PROGRAM PRG_KnxLine_1
  VAR
    M1_001_401_RMA6001_MOV_ACT : FbDPT_Switch_pro;
    M1_002_401_RMA6002_MOV_ACT : FbDPT_Switch_pro;
    M1_003_406_RMA6003_MOV_ACT : FbDPT_Switch_pro;
    M1_004_407_RMA6004_MOV_ACT : FbDPT_Switch_pro;
    M1_005_408_RMA6005_MOV_ACT : FbDPT_Switch_pro;
    M1_006_409_RMA6006_MOV_ACT : FbDPT_Switch_pro;
    M1_007_409_RMA6007_MOV_ACT : FbDPT_Switch_pro;
    M1_008_409_RMA6008_MOV_ACT : FbDPT_Switch_pro;
    M1_009_464_RMA6009_MOV_ACT : FbDPT_Switch_pro;
    M1_010_464_RMA6010_MOV_ACT : FbDPT_Switch_pro;
    M1_011_415_RMA6011_MOV_ACT : FbDPT_Switch_pro;
    M1_012_422_RMA6012_MOV_ACT : FbDPT_Switch_pro;
    M1_013_422_RMA6013_MOV_ACT : FbDPT_Switch_pro;
    M1_014_426_1_RMA6014_MOV_ACT : FbDPT_Switch_pro;
    M1_015_426_2_RMA6015_MOV_ACT : FbDPT_Switch_pro;
    M1_016_426_3_RMA6016_MOV_ACT : FbDPT_Switch_pro;
    M1_017_401_RMA6001_TMP_ACT : FbDPT_Value_Temp_pro;
    M1_018_401_RMA6002_TMP_ACT : FbDPT_Value_Temp_pro;
    M1_019_406_RMA6003_TMP_ACT : FbDPT_Value_Temp_pro;
    M1_020_407_RMA6004_TMP_ACT : FbDPT_Value_Temp_pro;
    M1_021_408_RMA6005_TMP_ACT : FbDPT_Value_Temp_pro;
    M1_022_409_RMA6006_TMP_ACT : FbDPT_Value_Temp_pro;
    M1_023_409_RMA6007_TMP_ACT : FbDPT_Value_Temp_pro;
    M1_024_409_RMA6008_TMP_ACT : FbDPT_Value_Temp_pro;
    M1_025_464_RMA6009_TMP_ACT : FbDPT_Value_Temp_pro;
    M1_026_464_RMA6010_TMP_ACT : FbDPT_Value_Temp_pro;
    M1_027_415_RMA6011_TMP_ACT : FbDPT_Value_Temp_pro;
    M1_028_422_RMA6012_TMP_ACT : FbDPT_Value_Temp_pro;
    M1_029_422_RMA6013_TMP_ACT : FbDPT_Value_Temp_pro;
    M1_030_426_1_RMA6014_TMP_ACT : FbDPT_Value_Temp_pro;
    M1_031_426_2_RMA6015_TMP_ACT : FbDPT_Value_Temp_pro;
    M1_032_426_3_RMA6016_TMP_ACT : FbDPT_Value_Temp_pro;
    M1_033_401_RMA6001_CO2_ACT : FbDPT_Value_AirQuality_pro;
    M1_034_401_RMA6002_CO2_ACT : FbDPT_Value_AirQuality_pro;
    M1_035_406_RMA6003_CO2_ACT : FbDPT_Value_AirQuality_pro;
    M1_036_407_RMA6004_CO2_ACT : FbDPT_Value_AirQuality_pro;
    M1_037_408_RMA6005_CO2_ACT : FbDPT_Value_AirQuality_pro;
    M1_038_409_RMA6006_CO2_ACT : FbDPT_Value_AirQuality_pro;
    M1_039_409_RMA6007_CO2_ACT : FbDPT_Value_AirQuality_pro;
    M1_040_409_RMA6008_CO2_ACT : FbDPT_Value_AirQuality_pro;
    M1_041_464_RMA6009_CO2_ACT : FbDPT_Value_AirQuality_pro;
    M1_042_464_RMA6010_CO2_ACT : FbDPT_Value_AirQuality_pro;
    M1_043_415_RMA6011_CO2_ACT : FbDPT_Value_AirQuality_pro;
    M1_044_422_RMA6012_CO2_ACT : FbDPT_Value_AirQuality_pro;
    M1_045_422_RMA6013_CO2_ACT : FbDPT_Value_AirQuality_pro;
    M1_046_426_1_RMA6014_CO2_ACT : FbDPT_Value_AirQuality_pro;
    M1_047_426_2_RMA6015_CO2_ACT : FbDPT_Value_AirQuality_pro;
    M1_048_426_3_RMA6016_CO2_ACT : FbDPT_Value_AirQuality_pro;
    M1_049_401_KAB6001_CV : FbDPT_Scaling_pro;
    M1_050_401_KAB6001_POS_ACT : FbDPT_Scaling_pro;
    M1_051_401_KAB6002_CV : FbDPT_Scaling_pro;
    M1_052_401_KAB6002_POS_ACT : FbDPT_Scaling_pro;
    M1_053_401_KAB6003_CV : FbDPT_Scaling_pro;
    M1_054_401_KAB6003_POS_ACT : FbDPT_Scaling_pro;
    M1_055_401_KAB6004_CV : FbDPT_Scaling_pro;
    M1_056_401_KAB6004_POS_ACT : FbDPT_Scaling_pro;
    M1_057_401_KAB6005_CV : FbDPT_Scaling_pro;
    M1_058_401_KAB6005_POS_ACT : FbDPT_Scaling_pro;
    M1_059_406_KAB6006_CV : FbDPT_Scaling_pro;
    M1_060_406_KAB6006_POS_ACT : FbDPT_Scaling_pro;
    M1_061_406_KAB6007_CV : FbDPT_Scaling_pro;
    M1_062_406_KAB6007_POS_ACT : FbDPT_Scaling_pro;
    M1_063_407_KAB6008_CV : FbDPT_Scaling_pro;
    M1_064_407_KAB6008_POS_ACT : FbDPT_Scaling_pro;
    M1_065_407_KAB6009_CV : FbDPT_Scaling_pro;
    M1_066_407_KAB6009_POS_ACT : FbDPT_Scaling_pro;
    M1_067_408_KAB6010_CV : FbDPT_Scaling_pro;
    M1_068_408_KAB6010_POS_ACT : FbDPT_Scaling_pro;
    M1_069_409_KAB6011_CV : FbDPT_Scaling_pro;
    M1_070_409_KAB6011_POS_ACT : FbDPT_Scaling_pro;
    M1_071_409_KAB6012_CV : FbDPT_Scaling_pro;
    M1_072_409_KAB6012_POS_ACT : FbDPT_Scaling_pro;
    M1_073_409_KAB6013_CV : FbDPT_Scaling_pro;
    M1_074_409_KAB6013_POS_ACT : FbDPT_Scaling_pro;
    M1_075_409_KAB6014_CV : FbDPT_Scaling_pro;
    M1_076_409_KAB6014_POS_ACT : FbDPT_Scaling_pro;
    M1_077_409_KAB6015_CV : FbDPT_Scaling_pro;
    M1_078_409_KAB6015_POS_ACT : FbDPT_Scaling_pro;
    M1_079_409_KAB6016_CV : FbDPT_Scaling_pro;
    M1_080_409_KAB6016_POS_ACT : FbDPT_Scaling_pro;
    M1_081_409_KAB6017_CV : FbDPT_Scaling_pro;
    M1_082_409_KAB6017_POS_ACT : FbDPT_Scaling_pro;
    M1_083_464_KAB6018_CV : FbDPT_Scaling_pro;
    M1_084_464_KAB6018_POS_ACT : FbDPT_Scaling_pro;
    M1_085_464_KAB6019_CV : FbDPT_Scaling_pro;
    M1_086_464_KAB6019_POS_ACT : FbDPT_Scaling_pro;
    M1_087_464_KAB6020_CV : FbDPT_Scaling_pro;
    M1_088_464_KAB6020_POS_ACT : FbDPT_Scaling_pro;
    M1_089_464_KAB6021_CV : FbDPT_Scaling_pro;
    M1_090_464_KAB6021_POS_ACT : FbDPT_Scaling_pro;
    M1_091_415_KAB6022_CV : FbDPT_Scaling_pro;
    M1_092_415_KAB6022_POS_ACT : FbDPT_Scaling_pro;
    M1_093_415_KAB6023_CV : FbDPT_Scaling_pro;
    M1_094_415_KAB6023_POS_ACT : FbDPT_Scaling_pro;
    M1_095_422_KAB6024_CV : FbDPT_Scaling_pro;
    M1_096_422_KAB6024_POS_ACT : FbDPT_Scaling_pro;
    M1_097_422_KAB6025_CV : FbDPT_Scaling_pro;
    M1_098_422_KAB6025_POS_ACT : FbDPT_Scaling_pro;
    M1_099_422_KAB6026_CV : FbDPT_Scaling_pro;
    M1_100_422_KAB6026_POS_ACT : FbDPT_Scaling_pro;
    M1_101_422_KAB6027_CV : FbDPT_Scaling_pro;
    M1_102_422_KAB6027_POS_ACT : FbDPT_Scaling_pro;
    M1_103_422_KAB6028_CV : FbDPT_Scaling_pro;
    M1_104_422_KAB6028_POS_ACT : FbDPT_Scaling_pro;
    M1_105_426_1_KAB6029_CV : FbDPT_Scaling_pro;
    M1_106_426_1_KAB6029_POS_ACT : FbDPT_Scaling_pro;
    M1_107_426_2_KAB6030_CV : FbDPT_Scaling_pro;
    M1_108_426_2_KAB6030_POS_ACT : FbDPT_Scaling_pro;
    M1_109_426_3_KAB6031_CV : FbDPT_Scaling_pro;
    M1_110_426_3_KAB6031_POS_ACT : FbDPT_Scaling_pro;
  END_VAR

                
    
        M1_001_401_RMA6001_MOV_ACT(
            bPortKNX      := 1, 
            dwIndex_DPT   := 1, 
            typDPT        := PersistentVars.typDPT[1][1]
        );

        
        M1_002_401_RMA6002_MOV_ACT(
            bPortKNX      := 1, 
            dwIndex_DPT   := 2, 
            typDPT        := PersistentVars.typDPT[1][2]
        );

        
        M1_003_406_RMA6003_MOV_ACT(
            bPortKNX      := 1, 
            dwIndex_DPT   := 3, 
            typDPT        := PersistentVars.typDPT[1][3]
        );

        
        M1_004_407_RMA6004_MOV_ACT(
            bPortKNX      := 1, 
            dwIndex_DPT   := 4, 
            typDPT        := PersistentVars.typDPT[1][4]
        );

        
        M1_005_408_RMA6005_MOV_ACT(
            bPortKNX      := 1, 
            dwIndex_DPT   := 5, 
            typDPT        := PersistentVars.typDPT[1][5]
        );

        
        M1_006_409_RMA6006_MOV_ACT(
            bPortKNX      := 1, 
            dwIndex_DPT   := 6, 
            typDPT        := PersistentVars.typDPT[1][6]
        );

        
        M1_007_409_RMA6007_MOV_ACT(
            bPortKNX      := 1, 
            dwIndex_DPT   := 7, 
            typDPT        := PersistentVars.typDPT[1][7]
        );

        
        M1_008_409_RMA6008_MOV_ACT(
            bPortKNX      := 1, 
            dwIndex_DPT   := 8, 
            typDPT        := PersistentVars.typDPT[1][8]
        );

        
        M1_009_464_RMA6009_MOV_ACT(
            bPortKNX      := 1, 
            dwIndex_DPT   := 9, 
            typDPT        := PersistentVars.typDPT[1][9]
        );

        
        M1_010_464_RMA6010_MOV_ACT(
            bPortKNX      := 1, 
            dwIndex_DPT   := 10, 
            typDPT        := PersistentVars.typDPT[1][10]
        );

        
        M1_011_415_RMA6011_MOV_ACT(
            bPortKNX      := 1, 
            dwIndex_DPT   := 11, 
            typDPT        := PersistentVars.typDPT[1][11]
        );

        
        M1_012_422_RMA6012_MOV_ACT(
            bPortKNX      := 1, 
            dwIndex_DPT   := 12, 
            typDPT        := PersistentVars.typDPT[1][12]
        );

        
        M1_013_422_RMA6013_MOV_ACT(
            bPortKNX      := 1, 
            dwIndex_DPT   := 13, 
            typDPT        := PersistentVars.typDPT[1][13]
        );

        
        M1_014_426_1_RMA6014_MOV_ACT(
            bPortKNX      := 1, 
            dwIndex_DPT   := 14, 
            typDPT        := PersistentVars.typDPT[1][14]
        );

        
        M1_015_426_2_RMA6015_MOV_ACT(
            bPortKNX      := 1, 
            dwIndex_DPT   := 15, 
            typDPT        := PersistentVars.typDPT[1][15]
        );

        
        M1_016_426_3_RMA6016_MOV_ACT(
            bPortKNX      := 1, 
            dwIndex_DPT   := 16, 
            typDPT        := PersistentVars.typDPT[1][16]
        );

        
        M1_017_401_RMA6001_TMP_ACT(
            bPortKNX      := 1,
            dwIndex_DPT   := 17,
            typDPT        := PersistentVars.typDPT[1][17],
            xUpdate_PLC   => ,
            xTimeOut      => 
        );

        
                                    
        C_5640_501_06_RMA6001_A1_R0401.xIn := M1_017_401_RMA6001_TMP_ACT.xTimeOut;
                                    
        M1_018_401_RMA6002_TMP_ACT(
            bPortKNX      := 1,
            dwIndex_DPT   := 18,
            typDPT        := PersistentVars.typDPT[1][18],
            xUpdate_PLC   => ,
            xTimeOut      => 
        );

        
                                    
        C_5640_501_06_RMA6002_A1_R0401.xIn := M1_018_401_RMA6002_TMP_ACT.xTimeOut;
                                    
        M1_019_406_RMA6003_TMP_ACT(
            bPortKNX      := 1,
            dwIndex_DPT   := 19,
            typDPT        := PersistentVars.typDPT[1][19],
            xUpdate_PLC   => ,
            xTimeOut      => 
        );

        
                                    
        C_5640_501_06_RMA6003_A1_R0406.xIn := M1_019_406_RMA6003_TMP_ACT.xTimeOut;
                                    
        M1_020_407_RMA6004_TMP_ACT(
            bPortKNX      := 1,
            dwIndex_DPT   := 20,
            typDPT        := PersistentVars.typDPT[1][20],
            xUpdate_PLC   => ,
            xTimeOut      => 
        );

        
                                    
        C_5640_501_06_RMA6004_A1_R0407.xIn := M1_020_407_RMA6004_TMP_ACT.xTimeOut;
                                    
        M1_021_408_RMA6005_TMP_ACT(
            bPortKNX      := 1,
            dwIndex_DPT   := 21,
            typDPT        := PersistentVars.typDPT[1][21],
            xUpdate_PLC   => ,
            xTimeOut      => 
        );

        
                                    
        C_5640_501_06_RMA6005_A1_R0408.xIn := M1_021_408_RMA6005_TMP_ACT.xTimeOut;
                                    
        M1_022_409_RMA6006_TMP_ACT(
            bPortKNX      := 1,
            dwIndex_DPT   := 22,
            typDPT        := PersistentVars.typDPT[1][22],
            xUpdate_PLC   => ,
            xTimeOut      => 
        );

        
                                    
        C_5640_501_06_RMA6006_A1_R0409.xIn := M1_022_409_RMA6006_TMP_ACT.xTimeOut;
                                    
        M1_023_409_RMA6007_TMP_ACT(
            bPortKNX      := 1,
            dwIndex_DPT   := 23,
            typDPT        := PersistentVars.typDPT[1][23],
            xUpdate_PLC   => ,
            xTimeOut      => 
        );

        
                                    
        C_5640_501_06_RMA6007_A1_R0409.xIn := M1_023_409_RMA6007_TMP_ACT.xTimeOut;
                                    
        M1_024_409_RMA6008_TMP_ACT(
            bPortKNX      := 1,
            dwIndex_DPT   := 24,
            typDPT        := PersistentVars.typDPT[1][24],
            xUpdate_PLC   => ,
            xTimeOut      => 
        );

        
                                    
        C_5640_501_06_RMA6008_A1_R0409.xIn := M1_024_409_RMA6008_TMP_ACT.xTimeOut;
                                    
        M1_025_464_RMA6009_TMP_ACT(
            bPortKNX      := 1,
            dwIndex_DPT   := 25,
            typDPT        := PersistentVars.typDPT[1][25],
            xUpdate_PLC   => ,
            xTimeOut      => 
        );

        
                                    
        C_5640_501_06_RMA6009_A1_R0464.xIn := M1_025_464_RMA6009_TMP_ACT.xTimeOut;
                                    
        M1_026_464_RMA6010_TMP_ACT(
            bPortKNX      := 1,
            dwIndex_DPT   := 26,
            typDPT        := PersistentVars.typDPT[1][26],
            xUpdate_PLC   => ,
            xTimeOut      => 
        );

        
                                    
        C_5640_501_06_RMA6010_A1_R0464.xIn := M1_026_464_RMA6010_TMP_ACT.xTimeOut;
                                    
        M1_027_415_RMA6011_TMP_ACT(
            bPortKNX      := 1,
            dwIndex_DPT   := 27,
            typDPT        := PersistentVars.typDPT[1][27],
            xUpdate_PLC   => ,
            xTimeOut      => 
        );

        
                                    
        C_5640_501_06_RMA6011_A1_R0415.xIn := M1_027_415_RMA6011_TMP_ACT.xTimeOut;
                                    
        M1_028_422_RMA6012_TMP_ACT(
            bPortKNX      := 1,
            dwIndex_DPT   := 28,
            typDPT        := PersistentVars.typDPT[1][28],
            xUpdate_PLC   => ,
            xTimeOut      => 
        );

        
                                    
        C_5640_501_06_RMA6012_A1_R0422.xIn := M1_028_422_RMA6012_TMP_ACT.xTimeOut;
                                    
        M1_029_422_RMA6013_TMP_ACT(
            bPortKNX      := 1,
            dwIndex_DPT   := 29,
            typDPT        := PersistentVars.typDPT[1][29],
            xUpdate_PLC   => ,
            xTimeOut      => 
        );

        
                                    
        C_5640_501_06_RMA6013_A1_R0422.xIn := M1_029_422_RMA6013_TMP_ACT.xTimeOut;
                                    
        M1_030_426_1_RMA6014_TMP_ACT(
            bPortKNX      := 1,
            dwIndex_DPT   := 30,
            typDPT        := PersistentVars.typDPT[1][30],
            xUpdate_PLC   => ,
            xTimeOut      => 
        );

        
                                    
        C_5640_501_06_RMA6014_A1_R0426_1.xIn := M1_030_426_1_RMA6014_TMP_ACT.xTimeOut;
                                    
        M1_031_426_2_RMA6015_TMP_ACT(
            bPortKNX      := 1,
            dwIndex_DPT   := 31,
            typDPT        := PersistentVars.typDPT[1][31],
            xUpdate_PLC   => ,
            xTimeOut      => 
        );

        
                                    
        C_5640_501_06_RMA6015_A1_R0426_2.xIn := M1_031_426_2_RMA6015_TMP_ACT.xTimeOut;
                                    
        M1_032_426_3_RMA6016_TMP_ACT(
            bPortKNX      := 1,
            dwIndex_DPT   := 32,
            typDPT        := PersistentVars.typDPT[1][32],
            xUpdate_PLC   => ,
            xTimeOut      => 
        );

        
                                    
        C_5640_501_06_RMA6016_A1_R0426_3.xIn := M1_032_426_3_RMA6016_TMP_ACT.xTimeOut;
                                    
        M1_033_401_RMA6001_CO2_ACT(
            bPortKNX      := 1,
            dwIndex_DPT   := 33,
            typDPT        := PersistentVars.typDPT[1][33],
            xUpdate_PLC   => ,
            xTimeOut      => 
        );

        
        M1_034_401_RMA6002_CO2_ACT(
            bPortKNX      := 1,
            dwIndex_DPT   := 34,
            typDPT        := PersistentVars.typDPT[1][34],
            xUpdate_PLC   => ,
            xTimeOut      => 
        );

        
        M1_035_406_RMA6003_CO2_ACT(
            bPortKNX      := 1,
            dwIndex_DPT   := 35,
            typDPT        := PersistentVars.typDPT[1][35],
            xUpdate_PLC   => ,
            xTimeOut      => 
        );

        
        M1_036_407_RMA6004_CO2_ACT(
            bPortKNX      := 1,
            dwIndex_DPT   := 36,
            typDPT        := PersistentVars.typDPT[1][36],
            xUpdate_PLC   => ,
            xTimeOut      => 
        );

        
        M1_037_408_RMA6005_CO2_ACT(
            bPortKNX      := 1,
            dwIndex_DPT   := 37,
            typDPT        := PersistentVars.typDPT[1][37],
            xUpdate_PLC   => ,
            xTimeOut      => 
        );

        
        M1_038_409_RMA6006_CO2_ACT(
            bPortKNX      := 1,
            dwIndex_DPT   := 38,
            typDPT        := PersistentVars.typDPT[1][38],
            xUpdate_PLC   => ,
            xTimeOut      => 
        );

        
        M1_039_409_RMA6007_CO2_ACT(
            bPortKNX      := 1,
            dwIndex_DPT   := 39,
            typDPT        := PersistentVars.typDPT[1][39],
            xUpdate_PLC   => ,
            xTimeOut      => 
        );

        
        M1_040_409_RMA6008_CO2_ACT(
            bPortKNX      := 1,
            dwIndex_DPT   := 40,
            typDPT        := PersistentVars.typDPT[1][40],
            xUpdate_PLC   => ,
            xTimeOut      => 
        );

        
        M1_041_464_RMA6009_CO2_ACT(
            bPortKNX      := 1,
            dwIndex_DPT   := 41,
            typDPT        := PersistentVars.typDPT[1][41],
            xUpdate_PLC   => ,
            xTimeOut      => 
        );

        
        M1_042_464_RMA6010_CO2_ACT(
            bPortKNX      := 1,
            dwIndex_DPT   := 42,
            typDPT        := PersistentVars.typDPT[1][42],
            xUpdate_PLC   => ,
            xTimeOut      => 
        );

        
        M1_043_415_RMA6011_CO2_ACT(
            bPortKNX      := 1,
            dwIndex_DPT   := 43,
            typDPT        := PersistentVars.typDPT[1][43],
            xUpdate_PLC   => ,
            xTimeOut      => 
        );

        
        M1_044_422_RMA6012_CO2_ACT(
            bPortKNX      := 1,
            dwIndex_DPT   := 44,
            typDPT        := PersistentVars.typDPT[1][44],
            xUpdate_PLC   => ,
            xTimeOut      => 
        );

        
        M1_045_422_RMA6013_CO2_ACT(
            bPortKNX      := 1,
            dwIndex_DPT   := 45,
            typDPT        := PersistentVars.typDPT[1][45],
            xUpdate_PLC   => ,
            xTimeOut      => 
        );

        
        M1_046_426_1_RMA6014_CO2_ACT(
            bPortKNX      := 1,
            dwIndex_DPT   := 46,
            typDPT        := PersistentVars.typDPT[1][46],
            xUpdate_PLC   => ,
            xTimeOut      => 
        );

        
        M1_047_426_2_RMA6015_CO2_ACT(
            bPortKNX      := 1,
            dwIndex_DPT   := 47,
            typDPT        := PersistentVars.typDPT[1][47],
            xUpdate_PLC   => ,
            xTimeOut      => 
        );

        
        M1_048_426_3_RMA6016_CO2_ACT(
            bPortKNX      := 1,
            dwIndex_DPT   := 48,
            typDPT        := PersistentVars.typDPT[1][48],
            xUpdate_PLC   => ,
            xTimeOut      => 
        );

        
        M1_049_401_KAB6001_CV(
            bPortKNX		  := 1, 
            dwIndex_DPT		:= 49, 
            typDPT			  := PersistentVars.typDPT[1][49],
            xUpdate_KNX		:= PRG_KnxMaster.updateHeat, 
        );

        M1_049_401_KAB6001_CV.rValue_IN := GVL_ClimateControl.typClimateControllerInterfaceRoom401.actuators.heating.controlledVariable;        
         
        M1_050_401_KAB6001_POS_ACT(
            bPortKNX		   := 1, 
            dwIndex_DPT		:= 50, 
            typDPT			  := PersistentVars.typDPT[1][50], 
        );

        
                                    
        C_5640_501_06_KAB6001_A1_R0401.xIn := M1_050_401_KAB6001_POS_ACT.xTimeOut;
                                    
        M1_051_401_KAB6002_CV(
            bPortKNX		  := 1, 
            dwIndex_DPT		:= 51, 
            typDPT			  := PersistentVars.typDPT[1][51],
            xUpdate_KNX		:= PRG_KnxMaster.updateHeat, 
        );

        M1_051_401_KAB6002_CV.rValue_IN := GVL_ClimateControl.typClimateControllerInterfaceRoom401.actuators.heating.controlledVariable;        
         
        M1_052_401_KAB6002_POS_ACT(
            bPortKNX		   := 1, 
            dwIndex_DPT		:= 52, 
            typDPT			  := PersistentVars.typDPT[1][52], 
        );

        
                                    
        C_5640_501_06_KAB6002_A1_R0401.xIn := M1_052_401_KAB6002_POS_ACT.xTimeOut;
                                    
        M1_053_401_KAB6003_CV(
            bPortKNX		  := 1, 
            dwIndex_DPT		:= 53, 
            typDPT			  := PersistentVars.typDPT[1][53],
            xUpdate_KNX		:= PRG_KnxMaster.updateHeat, 
        );

        M1_053_401_KAB6003_CV.rValue_IN := GVL_ClimateControl.typClimateControllerInterfaceRoom401.actuators.heating.controlledVariable;        
         
        M1_054_401_KAB6003_POS_ACT(
            bPortKNX		   := 1, 
            dwIndex_DPT		:= 54, 
            typDPT			  := PersistentVars.typDPT[1][54], 
        );

        
                                    
        C_5640_501_06_KAB6003_A1_R0401.xIn := M1_054_401_KAB6003_POS_ACT.xTimeOut;
                                    
        M1_055_401_KAB6004_CV(
            bPortKNX		  := 1, 
            dwIndex_DPT		:= 55, 
            typDPT			  := PersistentVars.typDPT[1][55],
            xUpdate_KNX		:= PRG_KnxMaster.updateHeat, 
        );

        M1_055_401_KAB6004_CV.rValue_IN := GVL_ClimateControl.typClimateControllerInterfaceRoom401.actuators.heating.controlledVariable;        
         
        M1_056_401_KAB6004_POS_ACT(
            bPortKNX		   := 1, 
            dwIndex_DPT		:= 56, 
            typDPT			  := PersistentVars.typDPT[1][56], 
        );

        
                                    
        C_5640_501_06_KAB6004_A1_R0401.xIn := M1_056_401_KAB6004_POS_ACT.xTimeOut;
                                    
        M1_057_401_KAB6005_CV(
            bPortKNX		  := 1, 
            dwIndex_DPT		:= 57, 
            typDPT			  := PersistentVars.typDPT[1][57],
            xUpdate_KNX		:= PRG_KnxMaster.updateHeat, 
        );

        M1_057_401_KAB6005_CV.rValue_IN := GVL_ClimateControl.typClimateControllerInterfaceRoom401.actuators.heating.controlledVariable;        
         
        M1_058_401_KAB6005_POS_ACT(
            bPortKNX		   := 1, 
            dwIndex_DPT		:= 58, 
            typDPT			  := PersistentVars.typDPT[1][58], 
        );

        
                                    
        C_5640_501_06_KAB6005_A1_R0401.xIn := M1_058_401_KAB6005_POS_ACT.xTimeOut;
                                    
        M1_059_406_KAB6006_CV(
            bPortKNX		  := 1, 
            dwIndex_DPT		:= 59, 
            typDPT			  := PersistentVars.typDPT[1][59],
            xUpdate_KNX		:= PRG_KnxMaster.updateHeat, 
        );

        M1_059_406_KAB6006_CV.rValue_IN := GVL_ClimateControl.typClimateControllerInterfaceRoom406.actuators.heating.controlledVariable;        
         
        M1_060_406_KAB6006_POS_ACT(
            bPortKNX		   := 1, 
            dwIndex_DPT		:= 60, 
            typDPT			  := PersistentVars.typDPT[1][60], 
        );

        
                                    
        C_5640_501_06_KAB6006_A1_R0406.xIn := M1_060_406_KAB6006_POS_ACT.xTimeOut;
                                    
        M1_061_406_KAB6007_CV(
            bPortKNX		  := 1, 
            dwIndex_DPT		:= 61, 
            typDPT			  := PersistentVars.typDPT[1][61],
            xUpdate_KNX		:= PRG_KnxMaster.updateHeat, 
        );

        M1_061_406_KAB6007_CV.rValue_IN := GVL_ClimateControl.typClimateControllerInterfaceRoom406.actuators.heating.controlledVariable;        
         
        M1_062_406_KAB6007_POS_ACT(
            bPortKNX		   := 1, 
            dwIndex_DPT		:= 62, 
            typDPT			  := PersistentVars.typDPT[1][62], 
        );

        
                                    
        C_5640_501_06_KAB6007_A1_R0406.xIn := M1_062_406_KAB6007_POS_ACT.xTimeOut;
                                    
        M1_063_407_KAB6008_CV(
            bPortKNX		  := 1, 
            dwIndex_DPT		:= 63, 
            typDPT			  := PersistentVars.typDPT[1][63],
            xUpdate_KNX		:= PRG_KnxMaster.updateHeat, 
        );

        M1_063_407_KAB6008_CV.rValue_IN := GVL_ClimateControl.typClimateControllerInterfaceRoom407.actuators.heating.controlledVariable;        
         
        M1_064_407_KAB6008_POS_ACT(
            bPortKNX		   := 1, 
            dwIndex_DPT		:= 64, 
            typDPT			  := PersistentVars.typDPT[1][64], 
        );

        
                                    
        C_5640_501_06_KAB6008_A1_R0407.xIn := M1_064_407_KAB6008_POS_ACT.xTimeOut;
                                    
        M1_065_407_KAB6009_CV(
            bPortKNX		  := 1, 
            dwIndex_DPT		:= 65, 
            typDPT			  := PersistentVars.typDPT[1][65],
            xUpdate_KNX		:= PRG_KnxMaster.updateHeat, 
        );

        M1_065_407_KAB6009_CV.rValue_IN := GVL_ClimateControl.typClimateControllerInterfaceRoom407.actuators.heating.controlledVariable;        
         
        M1_066_407_KAB6009_POS_ACT(
            bPortKNX		   := 1, 
            dwIndex_DPT		:= 66, 
            typDPT			  := PersistentVars.typDPT[1][66], 
        );

        
                                    
        C_5640_501_06_KAB6009_A1_R0407.xIn := M1_066_407_KAB6009_POS_ACT.xTimeOut;
                                    
        M1_067_408_KAB6010_CV(
            bPortKNX		  := 1, 
            dwIndex_DPT		:= 67, 
            typDPT			  := PersistentVars.typDPT[1][67],
            xUpdate_KNX		:= PRG_KnxMaster.updateHeat, 
        );

        M1_067_408_KAB6010_CV.rValue_IN := GVL_ClimateControl.typClimateControllerInterfaceRoom408.actuators.heating.controlledVariable;        
         
        M1_068_408_KAB6010_POS_ACT(
            bPortKNX		   := 1, 
            dwIndex_DPT		:= 68, 
            typDPT			  := PersistentVars.typDPT[1][68], 
        );

        
                                    
        C_5640_501_06_KAB6010_A1_R0408.xIn := M1_068_408_KAB6010_POS_ACT.xTimeOut;
                                    
        M1_069_409_KAB6011_CV(
            bPortKNX		  := 1, 
            dwIndex_DPT		:= 69, 
            typDPT			  := PersistentVars.typDPT[1][69],
            xUpdate_KNX		:= PRG_KnxMaster.updateHeat, 
        );

        M1_069_409_KAB6011_CV.rValue_IN := GVL_ClimateControl.typClimateControllerInterfaceRoom409.actuators.heating.controlledVariable;        
         
        M1_070_409_KAB6011_POS_ACT(
            bPortKNX		   := 1, 
            dwIndex_DPT		:= 70, 
            typDPT			  := PersistentVars.typDPT[1][70], 
        );

        
                                    
        C_5640_501_06_KAB6011_A1_R0409.xIn := M1_070_409_KAB6011_POS_ACT.xTimeOut;
                                    
        M1_071_409_KAB6012_CV(
            bPortKNX		  := 1, 
            dwIndex_DPT		:= 71, 
            typDPT			  := PersistentVars.typDPT[1][71],
            xUpdate_KNX		:= PRG_KnxMaster.updateHeat, 
        );

        M1_071_409_KAB6012_CV.rValue_IN := GVL_ClimateControl.typClimateControllerInterfaceRoom409.actuators.heating.controlledVariable;        
         
        M1_072_409_KAB6012_POS_ACT(
            bPortKNX		   := 1, 
            dwIndex_DPT		:= 72, 
            typDPT			  := PersistentVars.typDPT[1][72], 
        );

        
                                    
        C_5640_501_06_KAB6012_A1_R0409.xIn := M1_072_409_KAB6012_POS_ACT.xTimeOut;
                                    
        M1_073_409_KAB6013_CV(
            bPortKNX		  := 1, 
            dwIndex_DPT		:= 73, 
            typDPT			  := PersistentVars.typDPT[1][73],
            xUpdate_KNX		:= PRG_KnxMaster.updateHeat, 
        );

        M1_073_409_KAB6013_CV.rValue_IN := GVL_ClimateControl.typClimateControllerInterfaceRoom409.actuators.heating.controlledVariable;        
         
        M1_074_409_KAB6013_POS_ACT(
            bPortKNX		   := 1, 
            dwIndex_DPT		:= 74, 
            typDPT			  := PersistentVars.typDPT[1][74], 
        );

        
                                    
        C_5640_501_06_KAB6013_A1_R0409.xIn := M1_074_409_KAB6013_POS_ACT.xTimeOut;
                                    
        M1_075_409_KAB6014_CV(
            bPortKNX		  := 1, 
            dwIndex_DPT		:= 75, 
            typDPT			  := PersistentVars.typDPT[1][75],
            xUpdate_KNX		:= PRG_KnxMaster.updateHeat, 
        );

        M1_075_409_KAB6014_CV.rValue_IN := GVL_ClimateControl.typClimateControllerInterfaceRoom409.actuators.heating.controlledVariable;        
         
        M1_076_409_KAB6014_POS_ACT(
            bPortKNX		   := 1, 
            dwIndex_DPT		:= 76, 
            typDPT			  := PersistentVars.typDPT[1][76], 
        );

        
                                    
        C_5640_501_06_KAB6014_A1_R0409.xIn := M1_076_409_KAB6014_POS_ACT.xTimeOut;
                                    
        M1_077_409_KAB6015_CV(
            bPortKNX		  := 1, 
            dwIndex_DPT		:= 77, 
            typDPT			  := PersistentVars.typDPT[1][77],
            xUpdate_KNX		:= PRG_KnxMaster.updateHeat, 
        );

        M1_077_409_KAB6015_CV.rValue_IN := GVL_ClimateControl.typClimateControllerInterfaceRoom409.actuators.heating.controlledVariable;        
         
        M1_078_409_KAB6015_POS_ACT(
            bPortKNX		   := 1, 
            dwIndex_DPT		:= 78, 
            typDPT			  := PersistentVars.typDPT[1][78], 
        );

        
                                    
        C_5640_501_06_KAB6015_A1_R0409.xIn := M1_078_409_KAB6015_POS_ACT.xTimeOut;
                                    
        M1_079_409_KAB6016_CV(
            bPortKNX		  := 1, 
            dwIndex_DPT		:= 79, 
            typDPT			  := PersistentVars.typDPT[1][79],
            xUpdate_KNX		:= PRG_KnxMaster.updateHeat, 
        );

        M1_079_409_KAB6016_CV.rValue_IN := GVL_ClimateControl.typClimateControllerInterfaceRoom409.actuators.heating.controlledVariable;        
         
        M1_080_409_KAB6016_POS_ACT(
            bPortKNX		   := 1, 
            dwIndex_DPT		:= 80, 
            typDPT			  := PersistentVars.typDPT[1][80], 
        );

        
                                    
        C_5640_501_06_KAB6016_A1_R0409.xIn := M1_080_409_KAB6016_POS_ACT.xTimeOut;
                                    
        M1_081_409_KAB6017_CV(
            bPortKNX		  := 1, 
            dwIndex_DPT		:= 81, 
            typDPT			  := PersistentVars.typDPT[1][81],
            xUpdate_KNX		:= PRG_KnxMaster.updateHeat, 
        );

        M1_081_409_KAB6017_CV.rValue_IN := GVL_ClimateControl.typClimateControllerInterfaceRoom409.actuators.heating.controlledVariable;        
         
        M1_082_409_KAB6017_POS_ACT(
            bPortKNX		   := 1, 
            dwIndex_DPT		:= 82, 
            typDPT			  := PersistentVars.typDPT[1][82], 
        );

        
                                    
        C_5640_501_06_KAB6017_A1_R0409.xIn := M1_082_409_KAB6017_POS_ACT.xTimeOut;
                                    
        M1_083_464_KAB6018_CV(
            bPortKNX		  := 1, 
            dwIndex_DPT		:= 83, 
            typDPT			  := PersistentVars.typDPT[1][83],
            xUpdate_KNX		:= PRG_KnxMaster.updateHeat, 
        );

        M1_083_464_KAB6018_CV.rValue_IN := GVL_ClimateControl.typClimateControllerInterfaceRoom464.actuators.heating.controlledVariable;        
         
        M1_084_464_KAB6018_POS_ACT(
            bPortKNX		   := 1, 
            dwIndex_DPT		:= 84, 
            typDPT			  := PersistentVars.typDPT[1][84], 
        );

        
                                    
        C_5640_501_06_KAB6018_A1_R0464.xIn := M1_084_464_KAB6018_POS_ACT.xTimeOut;
                                    
        M1_085_464_KAB6019_CV(
            bPortKNX		  := 1, 
            dwIndex_DPT		:= 85, 
            typDPT			  := PersistentVars.typDPT[1][85],
            xUpdate_KNX		:= PRG_KnxMaster.updateHeat, 
        );

        M1_085_464_KAB6019_CV.rValue_IN := GVL_ClimateControl.typClimateControllerInterfaceRoom464.actuators.heating.controlledVariable;        
         
        M1_086_464_KAB6019_POS_ACT(
            bPortKNX		   := 1, 
            dwIndex_DPT		:= 86, 
            typDPT			  := PersistentVars.typDPT[1][86], 
        );

        
                                    
        C_5640_501_06_KAB6019_A1_R0464.xIn := M1_086_464_KAB6019_POS_ACT.xTimeOut;
                                    
        M1_087_464_KAB6020_CV(
            bPortKNX		  := 1, 
            dwIndex_DPT		:= 87, 
            typDPT			  := PersistentVars.typDPT[1][87],
            xUpdate_KNX		:= PRG_KnxMaster.updateHeat, 
        );

        M1_087_464_KAB6020_CV.rValue_IN := GVL_ClimateControl.typClimateControllerInterfaceRoom464.actuators.heating.controlledVariable;        
         
        M1_088_464_KAB6020_POS_ACT(
            bPortKNX		   := 1, 
            dwIndex_DPT		:= 88, 
            typDPT			  := PersistentVars.typDPT[1][88], 
        );

        
                                    
        C_5640_501_06_KAB6020_A1_R0464.xIn := M1_088_464_KAB6020_POS_ACT.xTimeOut;
                                    
        M1_089_464_KAB6021_CV(
            bPortKNX		  := 1, 
            dwIndex_DPT		:= 89, 
            typDPT			  := PersistentVars.typDPT[1][89],
            xUpdate_KNX		:= PRG_KnxMaster.updateHeat, 
        );

        M1_089_464_KAB6021_CV.rValue_IN := GVL_ClimateControl.typClimateControllerInterfaceRoom464.actuators.heating.controlledVariable;        
         
        M1_090_464_KAB6021_POS_ACT(
            bPortKNX		   := 1, 
            dwIndex_DPT		:= 90, 
            typDPT			  := PersistentVars.typDPT[1][90], 
        );

        
                                    
        C_5640_501_06_KAB6021_A1_R0464.xIn := M1_090_464_KAB6021_POS_ACT.xTimeOut;
                                    
        M1_091_415_KAB6022_CV(
            bPortKNX		  := 1, 
            dwIndex_DPT		:= 91, 
            typDPT			  := PersistentVars.typDPT[1][91],
            xUpdate_KNX		:= PRG_KnxMaster.updateHeat, 
        );

        M1_091_415_KAB6022_CV.rValue_IN := GVL_ClimateControl.typClimateControllerInterfaceRoom415.actuators.heating.controlledVariable;        
         
        M1_092_415_KAB6022_POS_ACT(
            bPortKNX		   := 1, 
            dwIndex_DPT		:= 92, 
            typDPT			  := PersistentVars.typDPT[1][92], 
        );

        
                                    
        C_5640_501_06_KAB6022_A1_R0415.xIn := M1_092_415_KAB6022_POS_ACT.xTimeOut;
                                    
        M1_093_415_KAB6023_CV(
            bPortKNX		  := 1, 
            dwIndex_DPT		:= 93, 
            typDPT			  := PersistentVars.typDPT[1][93],
            xUpdate_KNX		:= PRG_KnxMaster.updateHeat, 
        );

        M1_093_415_KAB6023_CV.rValue_IN := GVL_ClimateControl.typClimateControllerInterfaceRoom415.actuators.heating.controlledVariable;        
         
        M1_094_415_KAB6023_POS_ACT(
            bPortKNX		   := 1, 
            dwIndex_DPT		:= 94, 
            typDPT			  := PersistentVars.typDPT[1][94], 
        );

        
                                    
        C_5640_501_06_KAB6023_A1_R0415.xIn := M1_094_415_KAB6023_POS_ACT.xTimeOut;
                                    
        M1_095_422_KAB6024_CV(
            bPortKNX		  := 1, 
            dwIndex_DPT		:= 95, 
            typDPT			  := PersistentVars.typDPT[1][95],
            xUpdate_KNX		:= PRG_KnxMaster.updateHeat, 
        );

        M1_095_422_KAB6024_CV.rValue_IN := GVL_ClimateControl.typClimateControllerInterfaceRoom422.actuators.heating.controlledVariable;        
         
        M1_096_422_KAB6024_POS_ACT(
            bPortKNX		   := 1, 
            dwIndex_DPT		:= 96, 
            typDPT			  := PersistentVars.typDPT[1][96], 
        );

        
                                    
        C_5640_501_06_KAB6024_A1_R0422.xIn := M1_096_422_KAB6024_POS_ACT.xTimeOut;
                                    
        M1_097_422_KAB6025_CV(
            bPortKNX		  := 1, 
            dwIndex_DPT		:= 97, 
            typDPT			  := PersistentVars.typDPT[1][97],
            xUpdate_KNX		:= PRG_KnxMaster.updateHeat, 
        );

        M1_097_422_KAB6025_CV.rValue_IN := GVL_ClimateControl.typClimateControllerInterfaceRoom422.actuators.heating.controlledVariable;        
         
        M1_098_422_KAB6025_POS_ACT(
            bPortKNX		   := 1, 
            dwIndex_DPT		:= 98, 
            typDPT			  := PersistentVars.typDPT[1][98], 
        );

        
                                    
        C_5640_501_06_KAB6025_A1_R0422.xIn := M1_098_422_KAB6025_POS_ACT.xTimeOut;
                                    
        M1_099_422_KAB6026_CV(
            bPortKNX		  := 1, 
            dwIndex_DPT		:= 99, 
            typDPT			  := PersistentVars.typDPT[1][99],
            xUpdate_KNX		:= PRG_KnxMaster.updateHeat, 
        );

        M1_099_422_KAB6026_CV.rValue_IN := GVL_ClimateControl.typClimateControllerInterfaceRoom422.actuators.heating.controlledVariable;        
         
        M1_100_422_KAB6026_POS_ACT(
            bPortKNX		   := 1, 
            dwIndex_DPT		:= 100, 
            typDPT			  := PersistentVars.typDPT[1][100], 
        );

        
                                    
        C_5640_501_06_KAB6026_A1_R0422.xIn := M1_100_422_KAB6026_POS_ACT.xTimeOut;
                                    
        M1_101_422_KAB6027_CV(
            bPortKNX		  := 1, 
            dwIndex_DPT		:= 101, 
            typDPT			  := PersistentVars.typDPT[1][101],
            xUpdate_KNX		:= PRG_KnxMaster.updateHeat, 
        );

        M1_101_422_KAB6027_CV.rValue_IN := GVL_ClimateControl.typClimateControllerInterfaceRoom422.actuators.heating.controlledVariable;        
         
        M1_102_422_KAB6027_POS_ACT(
            bPortKNX		   := 1, 
            dwIndex_DPT		:= 102, 
            typDPT			  := PersistentVars.typDPT[1][102], 
        );

        
                                    
        C_5640_501_06_KAB6027_A1_R0422.xIn := M1_102_422_KAB6027_POS_ACT.xTimeOut;
                                    
        M1_103_422_KAB6028_CV(
            bPortKNX		  := 1, 
            dwIndex_DPT		:= 103, 
            typDPT			  := PersistentVars.typDPT[1][103],
            xUpdate_KNX		:= PRG_KnxMaster.updateHeat, 
        );

        M1_103_422_KAB6028_CV.rValue_IN := GVL_ClimateControl.typClimateControllerInterfaceRoom422.actuators.heating.controlledVariable;        
         
        M1_104_422_KAB6028_POS_ACT(
            bPortKNX		   := 1, 
            dwIndex_DPT		:= 104, 
            typDPT			  := PersistentVars.typDPT[1][104], 
        );

        
                                    
        C_5640_501_06_KAB6028_A1_R0422.xIn := M1_104_422_KAB6028_POS_ACT.xTimeOut;
                                    
        M1_105_426_1_KAB6029_CV(
            bPortKNX		  := 1, 
            dwIndex_DPT		:= 105, 
            typDPT			  := PersistentVars.typDPT[1][105],
            xUpdate_KNX		:= PRG_KnxMaster.updateHeat, 
        );

        M1_105_426_1_KAB6029_CV.rValue_IN := GVL_ClimateControl.typClimateControllerInterfaceRoom426_1.actuators.heating.controlledVariable;        
         
        M1_106_426_1_KAB6029_POS_ACT(
            bPortKNX		   := 1, 
            dwIndex_DPT		:= 106, 
            typDPT			  := PersistentVars.typDPT[1][106], 
        );

        
                                    
        C_5640_501_06_KAB6029_A1_R0426_1.xIn := M1_106_426_1_KAB6029_POS_ACT.xTimeOut;
                                    
        M1_107_426_2_KAB6030_CV(
            bPortKNX		  := 1, 
            dwIndex_DPT		:= 107, 
            typDPT			  := PersistentVars.typDPT[1][107],
            xUpdate_KNX		:= PRG_KnxMaster.updateHeat, 
        );

        M1_107_426_2_KAB6030_CV.rValue_IN := GVL_ClimateControl.typClimateControllerInterfaceRoom426_2.actuators.heating.controlledVariable;        
         
        M1_108_426_2_KAB6030_POS_ACT(
            bPortKNX		   := 1, 
            dwIndex_DPT		:= 108, 
            typDPT			  := PersistentVars.typDPT[1][108], 
        );

        
                                    
        C_5640_501_06_KAB6030_A1_R0426_2.xIn := M1_108_426_2_KAB6030_POS_ACT.xTimeOut;
                                    
        M1_109_426_3_KAB6031_CV(
            bPortKNX		  := 1, 
            dwIndex_DPT		:= 109, 
            typDPT			  := PersistentVars.typDPT[1][109],
            xUpdate_KNX		:= PRG_KnxMaster.updateHeat, 
        );

        M1_109_426_3_KAB6031_CV.rValue_IN := GVL_ClimateControl.typClimateControllerInterfaceRoom426_3.actuators.heating.controlledVariable;        
         
        M1_110_426_3_KAB6031_POS_ACT(
            bPortKNX		   := 1, 
            dwIndex_DPT		:= 110, 
            typDPT			  := PersistentVars.typDPT[1][110], 
        );

        
                                    
        C_5640_501_06_KAB6031_A1_R0426_3.xIn := M1_110_426_3_KAB6031_POS_ACT.xTimeOut;
                                    
                
              
END_PROGRAM

PROGRAM PRG_KnxLine_2
  VAR
    M2_001_528_RMA6001_MOV_ACT : FbDPT_Switch_pro;
    M2_002_523_RMA6002_MOV_ACT : FbDPT_Switch_pro;
    M2_003_531_RMA6003_MOV_ACT : FbDPT_Switch_pro;
    M2_004_535_1_RMA6004_MOV_ACT : FbDPT_Switch_pro;
    M2_005_535_2_RMA6005_MOV_ACT : FbDPT_Switch_pro;
    M2_006_535_3_RMA6006_MOV_ACT : FbDPT_Switch_pro;
    M2_007_536_RMA6007_MOV_ACT : FbDPT_Switch_pro;
    M2_008_543_RMA6008_MOV_ACT : FbDPT_Switch_pro;
    M2_009_547_1_RMA6009_MOV_ACT : FbDPT_Switch_pro;
    M2_010_547_2_RMA6010_MOV_ACT : FbDPT_Switch_pro;
    M2_011_544_RMA6011_MOV_ACT : FbDPT_Switch_pro;
    M2_012_544_RMA6012_MOV_ACT : FbDPT_Switch_pro;
    M2_013_528_RMA6001_TMP_ACT : FbDPT_Value_Temp_pro;
    M2_014_523_RMA6002_TMP_ACT : FbDPT_Value_Temp_pro;
    M2_015_531_RMA6003_TMP_ACT : FbDPT_Value_Temp_pro;
    M2_016_535_1_RMA6004_TMP_ACT : FbDPT_Value_Temp_pro;
    M2_017_535_2_RMA6005_TMP_ACT : FbDPT_Value_Temp_pro;
    M2_018_535_3_RMA6006_TMP_ACT : FbDPT_Value_Temp_pro;
    M2_019_536_RMA6007_TMP_ACT : FbDPT_Value_Temp_pro;
    M2_020_543_RMA6008_TMP_ACT : FbDPT_Value_Temp_pro;
    M2_021_547_1_RMA6009_TMP_ACT : FbDPT_Value_Temp_pro;
    M2_022_547_2_RMA6010_TMP_ACT : FbDPT_Value_Temp_pro;
    M2_023_544_RMA6011_TMP_ACT : FbDPT_Value_Temp_pro;
    M2_024_544_RMA6012_TMP_ACT : FbDPT_Value_Temp_pro;
    M2_025_528_RMA6001_CO2_ACT : FbDPT_Value_AirQuality_pro;
    M2_026_523_RMA6002_CO2_ACT : FbDPT_Value_AirQuality_pro;
    M2_027_531_RMA6003_CO2_ACT : FbDPT_Value_AirQuality_pro;
    M2_028_535_1_RMA6004_CO2_ACT : FbDPT_Value_AirQuality_pro;
    M2_029_535_2_RMA6005_CO2_ACT : FbDPT_Value_AirQuality_pro;
    M2_030_535_3_RMA6006_CO2_ACT : FbDPT_Value_AirQuality_pro;
    M2_031_536_RMA6007_CO2_ACT : FbDPT_Value_AirQuality_pro;
    M2_032_543_RMA6008_CO2_ACT : FbDPT_Value_AirQuality_pro;
    M2_033_547_1_RMA6009_CO2_ACT : FbDPT_Value_AirQuality_pro;
    M2_034_547_2_RMA6010_CO2_ACT : FbDPT_Value_AirQuality_pro;
    M2_035_544_RMA6011_CO2_ACT : FbDPT_Value_AirQuality_pro;
    M2_036_544_RMA6012_CO2_ACT : FbDPT_Value_AirQuality_pro;
    M2_037_528_KAB6001_CV : FbDPT_Scaling_pro;
    M2_038_528_KAB6001_POS_ACT : FbDPT_Scaling_pro;
    M2_039_523_KAB6002_CV : FbDPT_Scaling_pro;
    M2_040_523_KAB6002_POS_ACT : FbDPT_Scaling_pro;
    M2_041_531_KAB6003_CV : FbDPT_Scaling_pro;
    M2_042_531_KAB6003_POS_ACT : FbDPT_Scaling_pro;
    M2_043_531_KAB6004_CV : FbDPT_Scaling_pro;
    M2_044_531_KAB6004_POS_ACT : FbDPT_Scaling_pro;
    M2_045_535_1_KAB6005_CV : FbDPT_Scaling_pro;
    M2_046_535_1_KAB6005_POS_ACT : FbDPT_Scaling_pro;
    M2_047_535_1_KAB6006_CV : FbDPT_Scaling_pro;
    M2_048_535_1_KAB6006_POS_ACT : FbDPT_Scaling_pro;
    M2_049_535_1_KAB6007_CV : FbDPT_Scaling_pro;
    M2_050_535_1_KAB6007_POS_ACT : FbDPT_Scaling_pro;
    M2_051_535_1_KAB6008_CV : FbDPT_Scaling_pro;
    M2_052_535_1_KAB6008_POS_ACT : FbDPT_Scaling_pro;
    M2_053_535_2_KAB6009_CV : FbDPT_Scaling_pro;
    M2_054_535_2_KAB6009_POS_ACT : FbDPT_Scaling_pro;
    M2_055_535_2_KAB6010_CV : FbDPT_Scaling_pro;
    M2_056_535_2_KAB6010_POS_ACT : FbDPT_Scaling_pro;
    M2_057_535_2_KAB6011_CV : FbDPT_Scaling_pro;
    M2_058_535_2_KAB6011_POS_ACT : FbDPT_Scaling_pro;
    M2_059_535_2_KAB6012_CV : FbDPT_Scaling_pro;
    M2_060_535_2_KAB6012_POS_ACT : FbDPT_Scaling_pro;
    M2_061_535_2_KAB6013_CV : FbDPT_Scaling_pro;
    M2_062_535_2_KAB6013_POS_ACT : FbDPT_Scaling_pro;
    M2_063_535_2_KAB6014_CV : FbDPT_Scaling_pro;
    M2_064_535_2_KAB6014_POS_ACT : FbDPT_Scaling_pro;
    M2_065_535_3_KAB6015_CV : FbDPT_Scaling_pro;
    M2_066_535_3_KAB6015_POS_ACT : FbDPT_Scaling_pro;
    M2_067_535_3_KAB6016_CV : FbDPT_Scaling_pro;
    M2_068_535_3_KAB6016_POS_ACT : FbDPT_Scaling_pro;
    M2_069_535_3_KAB6017_CV : FbDPT_Scaling_pro;
    M2_070_535_3_KAB6017_POS_ACT : FbDPT_Scaling_pro;
    M2_071_536_KAB6018_CV : FbDPT_Scaling_pro;
    M2_072_536_KAB6018_POS_ACT : FbDPT_Scaling_pro;
    M2_073_536_KAB6019_CV : FbDPT_Scaling_pro;
    M2_074_536_KAB6019_POS_ACT : FbDPT_Scaling_pro;
    M2_075_543_KAB6020_CV : FbDPT_Scaling_pro;
    M2_076_543_KAB6020_POS_ACT : FbDPT_Scaling_pro;
    M2_077_543_KAB6021_CV : FbDPT_Scaling_pro;
    M2_078_543_KAB6021_POS_ACT : FbDPT_Scaling_pro;
    M2_079_547_1_KAB6022_CV : FbDPT_Scaling_pro;
    M2_080_547_1_KAB6022_POS_ACT : FbDPT_Scaling_pro;
    M2_081_547_1_KAB6023_CV : FbDPT_Scaling_pro;
    M2_082_547_1_KAB6023_POS_ACT : FbDPT_Scaling_pro;
    M2_083_547_1_KAB6024_CV : FbDPT_Scaling_pro;
    M2_084_547_1_KAB6024_POS_ACT : FbDPT_Scaling_pro;
    M2_085_547_2_KAB6025_CV : FbDPT_Scaling_pro;
    M2_086_547_2_KAB6025_POS_ACT : FbDPT_Scaling_pro;
    M2_087_547_2_KAB6026_CV : FbDPT_Scaling_pro;
    M2_088_547_2_KAB6026_POS_ACT : FbDPT_Scaling_pro;
    M2_089_547_2_KAB6027_CV : FbDPT_Scaling_pro;
    M2_090_547_2_KAB6027_POS_ACT : FbDPT_Scaling_pro;
    M2_091_544_KAB6028_CV : FbDPT_Scaling_pro;
    M2_092_544_KAB6028_POS_ACT : FbDPT_Scaling_pro;
  END_VAR

                
    
        M2_001_528_RMA6001_MOV_ACT(
            bPortKNX      := 2, 
            dwIndex_DPT   := 1, 
            typDPT        := PersistentVars.typDPT[2][1]
        );

        
        M2_002_523_RMA6002_MOV_ACT(
            bPortKNX      := 2, 
            dwIndex_DPT   := 2, 
            typDPT        := PersistentVars.typDPT[2][2]
        );

        
        M2_003_531_RMA6003_MOV_ACT(
            bPortKNX      := 2, 
            dwIndex_DPT   := 3, 
            typDPT        := PersistentVars.typDPT[2][3]
        );

        
        M2_004_535_1_RMA6004_MOV_ACT(
            bPortKNX      := 2, 
            dwIndex_DPT   := 4, 
            typDPT        := PersistentVars.typDPT[2][4]
        );

        
        M2_005_535_2_RMA6005_MOV_ACT(
            bPortKNX      := 2, 
            dwIndex_DPT   := 5, 
            typDPT        := PersistentVars.typDPT[2][5]
        );

        
        M2_006_535_3_RMA6006_MOV_ACT(
            bPortKNX      := 2, 
            dwIndex_DPT   := 6, 
            typDPT        := PersistentVars.typDPT[2][6]
        );

        
        M2_007_536_RMA6007_MOV_ACT(
            bPortKNX      := 2, 
            dwIndex_DPT   := 7, 
            typDPT        := PersistentVars.typDPT[2][7]
        );

        
        M2_008_543_RMA6008_MOV_ACT(
            bPortKNX      := 2, 
            dwIndex_DPT   := 8, 
            typDPT        := PersistentVars.typDPT[2][8]
        );

        
        M2_009_547_1_RMA6009_MOV_ACT(
            bPortKNX      := 2, 
            dwIndex_DPT   := 9, 
            typDPT        := PersistentVars.typDPT[2][9]
        );

        
        M2_010_547_2_RMA6010_MOV_ACT(
            bPortKNX      := 2, 
            dwIndex_DPT   := 10, 
            typDPT        := PersistentVars.typDPT[2][10]
        );

        
        M2_011_544_RMA6011_MOV_ACT(
            bPortKNX      := 2, 
            dwIndex_DPT   := 11, 
            typDPT        := PersistentVars.typDPT[2][11]
        );

        
        M2_012_544_RMA6012_MOV_ACT(
            bPortKNX      := 2, 
            dwIndex_DPT   := 12, 
            typDPT        := PersistentVars.typDPT[2][12]
        );

        
        M2_013_528_RMA6001_TMP_ACT(
            bPortKNX      := 2,
            dwIndex_DPT   := 13,
            typDPT        := PersistentVars.typDPT[2][13],
            xUpdate_PLC   => ,
            xTimeOut      => 
        );

        
                                    
        C_5640_501_06_RMA6001_A1_R0528.xIn := M2_013_528_RMA6001_TMP_ACT.xTimeOut;
                                    
        M2_014_523_RMA6002_TMP_ACT(
            bPortKNX      := 2,
            dwIndex_DPT   := 14,
            typDPT        := PersistentVars.typDPT[2][14],
            xUpdate_PLC   => ,
            xTimeOut      => 
        );

        
                                    
        C_5640_501_06_RMA6002_A1_R0523.xIn := M2_014_523_RMA6002_TMP_ACT.xTimeOut;
                                    
        M2_015_531_RMA6003_TMP_ACT(
            bPortKNX      := 2,
            dwIndex_DPT   := 15,
            typDPT        := PersistentVars.typDPT[2][15],
            xUpdate_PLC   => ,
            xTimeOut      => 
        );

        
                                    
        C_5640_501_06_RMA6003_A1_R0531.xIn := M2_015_531_RMA6003_TMP_ACT.xTimeOut;
                                    
        M2_016_535_1_RMA6004_TMP_ACT(
            bPortKNX      := 2,
            dwIndex_DPT   := 16,
            typDPT        := PersistentVars.typDPT[2][16],
            xUpdate_PLC   => ,
            xTimeOut      => 
        );

        
                                    
        C_5640_501_06_RMA6004_A1_R0535_1.xIn := M2_016_535_1_RMA6004_TMP_ACT.xTimeOut;
                                    
        M2_017_535_2_RMA6005_TMP_ACT(
            bPortKNX      := 2,
            dwIndex_DPT   := 17,
            typDPT        := PersistentVars.typDPT[2][17],
            xUpdate_PLC   => ,
            xTimeOut      => 
        );

        
                                    
        C_5640_501_06_RMA6005_A1_R0535_2.xIn := M2_017_535_2_RMA6005_TMP_ACT.xTimeOut;
                                    
        M2_018_535_3_RMA6006_TMP_ACT(
            bPortKNX      := 2,
            dwIndex_DPT   := 18,
            typDPT        := PersistentVars.typDPT[2][18],
            xUpdate_PLC   => ,
            xTimeOut      => 
        );

        
                                    
        C_5640_501_06_RMA6006_A1_R0535_3.xIn := M2_018_535_3_RMA6006_TMP_ACT.xTimeOut;
                                    
        M2_019_536_RMA6007_TMP_ACT(
            bPortKNX      := 2,
            dwIndex_DPT   := 19,
            typDPT        := PersistentVars.typDPT[2][19],
            xUpdate_PLC   => ,
            xTimeOut      => 
        );

        
                                    
        C_5640_501_06_RMA6007_A1_R0536.xIn := M2_019_536_RMA6007_TMP_ACT.xTimeOut;
                                    
        M2_020_543_RMA6008_TMP_ACT(
            bPortKNX      := 2,
            dwIndex_DPT   := 20,
            typDPT        := PersistentVars.typDPT[2][20],
            xUpdate_PLC   => ,
            xTimeOut      => 
        );

        
                                    
        C_5640_501_06_RMA6008_A1_R0543.xIn := M2_020_543_RMA6008_TMP_ACT.xTimeOut;
                                    
        M2_021_547_1_RMA6009_TMP_ACT(
            bPortKNX      := 2,
            dwIndex_DPT   := 21,
            typDPT        := PersistentVars.typDPT[2][21],
            xUpdate_PLC   => ,
            xTimeOut      => 
        );

        
                                    
        C_5640_501_06_RMA6009_A1_R0547_1.xIn := M2_021_547_1_RMA6009_TMP_ACT.xTimeOut;
                                    
        M2_022_547_2_RMA6010_TMP_ACT(
            bPortKNX      := 2,
            dwIndex_DPT   := 22,
            typDPT        := PersistentVars.typDPT[2][22],
            xUpdate_PLC   => ,
            xTimeOut      => 
        );

        
                                    
        C_5640_501_06_RMA6010_A1_R0547_2.xIn := M2_022_547_2_RMA6010_TMP_ACT.xTimeOut;
                                    
        M2_023_544_RMA6011_TMP_ACT(
            bPortKNX      := 2,
            dwIndex_DPT   := 23,
            typDPT        := PersistentVars.typDPT[2][23],
            xUpdate_PLC   => ,
            xTimeOut      => 
        );

        
                                    
        C_5640_501_06_RMA6011_A1_R0544.xIn := M2_023_544_RMA6011_TMP_ACT.xTimeOut;
                                    
        M2_024_544_RMA6012_TMP_ACT(
            bPortKNX      := 2,
            dwIndex_DPT   := 24,
            typDPT        := PersistentVars.typDPT[2][24],
            xUpdate_PLC   => ,
            xTimeOut      => 
        );

        
                                    
        C_5640_501_06_RMA6012_A1_R0544.xIn := M2_024_544_RMA6012_TMP_ACT.xTimeOut;
                                    
        M2_025_528_RMA6001_CO2_ACT(
            bPortKNX      := 2,
            dwIndex_DPT   := 25,
            typDPT        := PersistentVars.typDPT[2][25],
            xUpdate_PLC   => ,
            xTimeOut      => 
        );

        
        M2_026_523_RMA6002_CO2_ACT(
            bPortKNX      := 2,
            dwIndex_DPT   := 26,
            typDPT        := PersistentVars.typDPT[2][26],
            xUpdate_PLC   => ,
            xTimeOut      => 
        );

        
        M2_027_531_RMA6003_CO2_ACT(
            bPortKNX      := 2,
            dwIndex_DPT   := 27,
            typDPT        := PersistentVars.typDPT[2][27],
            xUpdate_PLC   => ,
            xTimeOut      => 
        );

        
        M2_028_535_1_RMA6004_CO2_ACT(
            bPortKNX      := 2,
            dwIndex_DPT   := 28,
            typDPT        := PersistentVars.typDPT[2][28],
            xUpdate_PLC   => ,
            xTimeOut      => 
        );

        
        M2_029_535_2_RMA6005_CO2_ACT(
            bPortKNX      := 2,
            dwIndex_DPT   := 29,
            typDPT        := PersistentVars.typDPT[2][29],
            xUpdate_PLC   => ,
            xTimeOut      => 
        );

        
        M2_030_535_3_RMA6006_CO2_ACT(
            bPortKNX      := 2,
            dwIndex_DPT   := 30,
            typDPT        := PersistentVars.typDPT[2][30],
            xUpdate_PLC   => ,
            xTimeOut      => 
        );

        
        M2_031_536_RMA6007_CO2_ACT(
            bPortKNX      := 2,
            dwIndex_DPT   := 31,
            typDPT        := PersistentVars.typDPT[2][31],
            xUpdate_PLC   => ,
            xTimeOut      => 
        );

        
        M2_032_543_RMA6008_CO2_ACT(
            bPortKNX      := 2,
            dwIndex_DPT   := 32,
            typDPT        := PersistentVars.typDPT[2][32],
            xUpdate_PLC   => ,
            xTimeOut      => 
        );

        
        M2_033_547_1_RMA6009_CO2_ACT(
            bPortKNX      := 2,
            dwIndex_DPT   := 33,
            typDPT        := PersistentVars.typDPT[2][33],
            xUpdate_PLC   => ,
            xTimeOut      => 
        );

        
        M2_034_547_2_RMA6010_CO2_ACT(
            bPortKNX      := 2,
            dwIndex_DPT   := 34,
            typDPT        := PersistentVars.typDPT[2][34],
            xUpdate_PLC   => ,
            xTimeOut      => 
        );

        
        M2_035_544_RMA6011_CO2_ACT(
            bPortKNX      := 2,
            dwIndex_DPT   := 35,
            typDPT        := PersistentVars.typDPT[2][35],
            xUpdate_PLC   => ,
            xTimeOut      => 
        );

        
        M2_036_544_RMA6012_CO2_ACT(
            bPortKNX      := 2,
            dwIndex_DPT   := 36,
            typDPT        := PersistentVars.typDPT[2][36],
            xUpdate_PLC   => ,
            xTimeOut      => 
        );

        
        M2_037_528_KAB6001_CV(
            bPortKNX		  := 2, 
            dwIndex_DPT		:= 37, 
            typDPT			  := PersistentVars.typDPT[2][37],
            xUpdate_KNX		:= PRG_KnxMaster.updateHeat, 
        );

        M2_037_528_KAB6001_CV.rValue_IN := GVL_ClimateControl.typClimateControllerInterfaceRoom528.actuators.heating.controlledVariable;        
         
        M2_038_528_KAB6001_POS_ACT(
            bPortKNX		   := 2, 
            dwIndex_DPT		:= 38, 
            typDPT			  := PersistentVars.typDPT[2][38], 
        );

        
                                    
        C_5640_501_06_KAB6001_A1_R0528.xIn := M2_038_528_KAB6001_POS_ACT.xTimeOut;
                                    
        M2_039_523_KAB6002_CV(
            bPortKNX		  := 2, 
            dwIndex_DPT		:= 39, 
            typDPT			  := PersistentVars.typDPT[2][39],
            xUpdate_KNX		:= PRG_KnxMaster.updateHeat, 
        );

        M2_039_523_KAB6002_CV.rValue_IN := GVL_ClimateControl.typClimateControllerInterfaceRoom523.actuators.heating.controlledVariable;        
         
        M2_040_523_KAB6002_POS_ACT(
            bPortKNX		   := 2, 
            dwIndex_DPT		:= 40, 
            typDPT			  := PersistentVars.typDPT[2][40], 
        );

        
                                    
        C_5640_501_06_KAB6002_A1_R0523.xIn := M2_040_523_KAB6002_POS_ACT.xTimeOut;
                                    
        M2_041_531_KAB6003_CV(
            bPortKNX		  := 2, 
            dwIndex_DPT		:= 41, 
            typDPT			  := PersistentVars.typDPT[2][41],
            xUpdate_KNX		:= PRG_KnxMaster.updateHeat, 
        );

        M2_041_531_KAB6003_CV.rValue_IN := GVL_ClimateControl.typClimateControllerInterfaceRoom531.actuators.heating.controlledVariable;        
         
        M2_042_531_KAB6003_POS_ACT(
            bPortKNX		   := 2, 
            dwIndex_DPT		:= 42, 
            typDPT			  := PersistentVars.typDPT[2][42], 
        );

        
                                    
        C_5640_501_06_KAB6003_A1_R0531.xIn := M2_042_531_KAB6003_POS_ACT.xTimeOut;
                                    
        M2_043_531_KAB6004_CV(
            bPortKNX		  := 2, 
            dwIndex_DPT		:= 43, 
            typDPT			  := PersistentVars.typDPT[2][43],
            xUpdate_KNX		:= PRG_KnxMaster.updateHeat, 
        );

        M2_043_531_KAB6004_CV.rValue_IN := GVL_ClimateControl.typClimateControllerInterfaceRoom531.actuators.heating.controlledVariable;        
         
        M2_044_531_KAB6004_POS_ACT(
            bPortKNX		   := 2, 
            dwIndex_DPT		:= 44, 
            typDPT			  := PersistentVars.typDPT[2][44], 
        );

        
                                    
        C_5640_501_06_KAB6004_A1_R0531.xIn := M2_044_531_KAB6004_POS_ACT.xTimeOut;
                                    
        M2_045_535_1_KAB6005_CV(
            bPortKNX		  := 2, 
            dwIndex_DPT		:= 45, 
            typDPT			  := PersistentVars.typDPT[2][45],
            xUpdate_KNX		:= PRG_KnxMaster.updateHeat, 
        );

        M2_045_535_1_KAB6005_CV.rValue_IN := GVL_ClimateControl.typClimateControllerInterfaceRoom535_1.actuators.heating.controlledVariable;        
         
        M2_046_535_1_KAB6005_POS_ACT(
            bPortKNX		   := 2, 
            dwIndex_DPT		:= 46, 
            typDPT			  := PersistentVars.typDPT[2][46], 
        );

        
                                    
        C_5640_501_06_KAB6005_A1_R0535_1.xIn := M2_046_535_1_KAB6005_POS_ACT.xTimeOut;
                                    
        M2_047_535_1_KAB6006_CV(
            bPortKNX		  := 2, 
            dwIndex_DPT		:= 47, 
            typDPT			  := PersistentVars.typDPT[2][47],
            xUpdate_KNX		:= PRG_KnxMaster.updateHeat, 
        );

        M2_047_535_1_KAB6006_CV.rValue_IN := GVL_ClimateControl.typClimateControllerInterfaceRoom535_1.actuators.heating.controlledVariable;        
         
        M2_048_535_1_KAB6006_POS_ACT(
            bPortKNX		   := 2, 
            dwIndex_DPT		:= 48, 
            typDPT			  := PersistentVars.typDPT[2][48], 
        );

        
                                    
        C_5640_501_06_KAB6006_A1_R0535_1.xIn := M2_048_535_1_KAB6006_POS_ACT.xTimeOut;
                                    
        M2_049_535_1_KAB6007_CV(
            bPortKNX		  := 2, 
            dwIndex_DPT		:= 49, 
            typDPT			  := PersistentVars.typDPT[2][49],
            xUpdate_KNX		:= PRG_KnxMaster.updateHeat, 
        );

        M2_049_535_1_KAB6007_CV.rValue_IN := GVL_ClimateControl.typClimateControllerInterfaceRoom535_1.actuators.heating.controlledVariable;        
         
        M2_050_535_1_KAB6007_POS_ACT(
            bPortKNX		   := 2, 
            dwIndex_DPT		:= 50, 
            typDPT			  := PersistentVars.typDPT[2][50], 
        );

        
                                    
        C_5640_501_06_KAB6007_A1_R0535_1.xIn := M2_050_535_1_KAB6007_POS_ACT.xTimeOut;
                                    
        M2_051_535_1_KAB6008_CV(
            bPortKNX		  := 2, 
            dwIndex_DPT		:= 51, 
            typDPT			  := PersistentVars.typDPT[2][51],
            xUpdate_KNX		:= PRG_KnxMaster.updateHeat, 
        );

        M2_051_535_1_KAB6008_CV.rValue_IN := GVL_ClimateControl.typClimateControllerInterfaceRoom535_1.actuators.heating.controlledVariable;        
         
        M2_052_535_1_KAB6008_POS_ACT(
            bPortKNX		   := 2, 
            dwIndex_DPT		:= 52, 
            typDPT			  := PersistentVars.typDPT[2][52], 
        );

        
                                    
        C_5640_501_06_KAB6008_A1_R0535_1.xIn := M2_052_535_1_KAB6008_POS_ACT.xTimeOut;
                                    
        M2_053_535_2_KAB6009_CV(
            bPortKNX		  := 2, 
            dwIndex_DPT		:= 53, 
            typDPT			  := PersistentVars.typDPT[2][53],
            xUpdate_KNX		:= PRG_KnxMaster.updateHeat, 
        );

        M2_053_535_2_KAB6009_CV.rValue_IN := GVL_ClimateControl.typClimateControllerInterfaceRoom535_2.actuators.heating.controlledVariable;        
         
        M2_054_535_2_KAB6009_POS_ACT(
            bPortKNX		   := 2, 
            dwIndex_DPT		:= 54, 
            typDPT			  := PersistentVars.typDPT[2][54], 
        );

        
                                    
        C_5640_501_06_KAB6009_A1_R0535_2.xIn := M2_054_535_2_KAB6009_POS_ACT.xTimeOut;
                                    
        M2_055_535_2_KAB6010_CV(
            bPortKNX		  := 2, 
            dwIndex_DPT		:= 55, 
            typDPT			  := PersistentVars.typDPT[2][55],
            xUpdate_KNX		:= PRG_KnxMaster.updateHeat, 
        );

        M2_055_535_2_KAB6010_CV.rValue_IN := GVL_ClimateControl.typClimateControllerInterfaceRoom535_2.actuators.heating.controlledVariable;        
         
        M2_056_535_2_KAB6010_POS_ACT(
            bPortKNX		   := 2, 
            dwIndex_DPT		:= 56, 
            typDPT			  := PersistentVars.typDPT[2][56], 
        );

        
                                    
        C_5640_501_06_KAB6010_A1_R0535_2.xIn := M2_056_535_2_KAB6010_POS_ACT.xTimeOut;
                                    
        M2_057_535_2_KAB6011_CV(
            bPortKNX		  := 2, 
            dwIndex_DPT		:= 57, 
            typDPT			  := PersistentVars.typDPT[2][57],
            xUpdate_KNX		:= PRG_KnxMaster.updateHeat, 
        );

        M2_057_535_2_KAB6011_CV.rValue_IN := GVL_ClimateControl.typClimateControllerInterfaceRoom535_2.actuators.heating.controlledVariable;        
         
        M2_058_535_2_KAB6011_POS_ACT(
            bPortKNX		   := 2, 
            dwIndex_DPT		:= 58, 
            typDPT			  := PersistentVars.typDPT[2][58], 
        );

        
                                    
        C_5640_501_06_KAB6011_A1_R0535_2.xIn := M2_058_535_2_KAB6011_POS_ACT.xTimeOut;
                                    
        M2_059_535_2_KAB6012_CV(
            bPortKNX		  := 2, 
            dwIndex_DPT		:= 59, 
            typDPT			  := PersistentVars.typDPT[2][59],
            xUpdate_KNX		:= PRG_KnxMaster.updateHeat, 
        );

        M2_059_535_2_KAB6012_CV.rValue_IN := GVL_ClimateControl.typClimateControllerInterfaceRoom535_2.actuators.heating.controlledVariable;        
         
        M2_060_535_2_KAB6012_POS_ACT(
            bPortKNX		   := 2, 
            dwIndex_DPT		:= 60, 
            typDPT			  := PersistentVars.typDPT[2][60], 
        );

        
                                    
        C_5640_501_06_KAB6012_A1_R0535_2.xIn := M2_060_535_2_KAB6012_POS_ACT.xTimeOut;
                                    
        M2_061_535_2_KAB6013_CV(
            bPortKNX		  := 2, 
            dwIndex_DPT		:= 61, 
            typDPT			  := PersistentVars.typDPT[2][61],
            xUpdate_KNX		:= PRG_KnxMaster.updateHeat, 
        );

        M2_061_535_2_KAB6013_CV.rValue_IN := GVL_ClimateControl.typClimateControllerInterfaceRoom535_2.actuators.heating.controlledVariable;        
         
        M2_062_535_2_KAB6013_POS_ACT(
            bPortKNX		   := 2, 
            dwIndex_DPT		:= 62, 
            typDPT			  := PersistentVars.typDPT[2][62], 
        );

        
                                    
        C_5640_501_06_KAB6013_A1_R0535_2.xIn := M2_062_535_2_KAB6013_POS_ACT.xTimeOut;
                                    
        M2_063_535_2_KAB6014_CV(
            bPortKNX		  := 2, 
            dwIndex_DPT		:= 63, 
            typDPT			  := PersistentVars.typDPT[2][63],
            xUpdate_KNX		:= PRG_KnxMaster.updateHeat, 
        );

        M2_063_535_2_KAB6014_CV.rValue_IN := GVL_ClimateControl.typClimateControllerInterfaceRoom535_2.actuators.heating.controlledVariable;        
         
        M2_064_535_2_KAB6014_POS_ACT(
            bPortKNX		   := 2, 
            dwIndex_DPT		:= 64, 
            typDPT			  := PersistentVars.typDPT[2][64], 
        );

        
                                    
        C_5640_501_06_KAB6014_A1_R0535_2.xIn := M2_064_535_2_KAB6014_POS_ACT.xTimeOut;
                                    
        M2_065_535_3_KAB6015_CV(
            bPortKNX		  := 2, 
            dwIndex_DPT		:= 65, 
            typDPT			  := PersistentVars.typDPT[2][65],
            xUpdate_KNX		:= PRG_KnxMaster.updateHeat, 
        );

        M2_065_535_3_KAB6015_CV.rValue_IN := GVL_ClimateControl.typClimateControllerInterfaceRoom535_3.actuators.heating.controlledVariable;        
         
        M2_066_535_3_KAB6015_POS_ACT(
            bPortKNX		   := 2, 
            dwIndex_DPT		:= 66, 
            typDPT			  := PersistentVars.typDPT[2][66], 
        );

        
                                    
        C_5640_501_06_KAB6015_A1_R0535_3.xIn := M2_066_535_3_KAB6015_POS_ACT.xTimeOut;
                                    
        M2_067_535_3_KAB6016_CV(
            bPortKNX		  := 2, 
            dwIndex_DPT		:= 67, 
            typDPT			  := PersistentVars.typDPT[2][67],
            xUpdate_KNX		:= PRG_KnxMaster.updateHeat, 
        );

        M2_067_535_3_KAB6016_CV.rValue_IN := GVL_ClimateControl.typClimateControllerInterfaceRoom535_3.actuators.heating.controlledVariable;        
         
        M2_068_535_3_KAB6016_POS_ACT(
            bPortKNX		   := 2, 
            dwIndex_DPT		:= 68, 
            typDPT			  := PersistentVars.typDPT[2][68], 
        );

        
                                    
        C_5640_501_06_KAB6016_A1_R0535_3.xIn := M2_068_535_3_KAB6016_POS_ACT.xTimeOut;
                                    
        M2_069_535_3_KAB6017_CV(
            bPortKNX		  := 2, 
            dwIndex_DPT		:= 69, 
            typDPT			  := PersistentVars.typDPT[2][69],
            xUpdate_KNX		:= PRG_KnxMaster.updateHeat, 
        );

        M2_069_535_3_KAB6017_CV.rValue_IN := GVL_ClimateControl.typClimateControllerInterfaceRoom535_3.actuators.heating.controlledVariable;        
         
        M2_070_535_3_KAB6017_POS_ACT(
            bPortKNX		   := 2, 
            dwIndex_DPT		:= 70, 
            typDPT			  := PersistentVars.typDPT[2][70], 
        );

        
                                    
        C_5640_501_06_KAB6017_A1_R0535_3.xIn := M2_070_535_3_KAB6017_POS_ACT.xTimeOut;
                                    
        M2_071_536_KAB6018_CV(
            bPortKNX		  := 2, 
            dwIndex_DPT		:= 71, 
            typDPT			  := PersistentVars.typDPT[2][71],
            xUpdate_KNX		:= PRG_KnxMaster.updateHeat, 
        );

        M2_071_536_KAB6018_CV.rValue_IN := GVL_ClimateControl.typClimateControllerInterfaceRoom536.actuators.heating.controlledVariable;        
         
        M2_072_536_KAB6018_POS_ACT(
            bPortKNX		   := 2, 
            dwIndex_DPT		:= 72, 
            typDPT			  := PersistentVars.typDPT[2][72], 
        );

        
                                    
        C_5640_501_06_KAB6018_A1_R0536.xIn := M2_072_536_KAB6018_POS_ACT.xTimeOut;
                                    
        M2_073_536_KAB6019_CV(
            bPortKNX		  := 2, 
            dwIndex_DPT		:= 73, 
            typDPT			  := PersistentVars.typDPT[2][73],
            xUpdate_KNX		:= PRG_KnxMaster.updateHeat, 
        );

        M2_073_536_KAB6019_CV.rValue_IN := GVL_ClimateControl.typClimateControllerInterfaceRoom536.actuators.heating.controlledVariable;        
         
        M2_074_536_KAB6019_POS_ACT(
            bPortKNX		   := 2, 
            dwIndex_DPT		:= 74, 
            typDPT			  := PersistentVars.typDPT[2][74], 
        );

        
                                    
        C_5640_501_06_KAB6019_A1_R0536.xIn := M2_074_536_KAB6019_POS_ACT.xTimeOut;
                                    
        M2_075_543_KAB6020_CV(
            bPortKNX		  := 2, 
            dwIndex_DPT		:= 75, 
            typDPT			  := PersistentVars.typDPT[2][75],
            xUpdate_KNX		:= PRG_KnxMaster.updateHeat, 
        );

        M2_075_543_KAB6020_CV.rValue_IN := GVL_ClimateControl.typClimateControllerInterfaceRoom543.actuators.heating.controlledVariable;        
         
        M2_076_543_KAB6020_POS_ACT(
            bPortKNX		   := 2, 
            dwIndex_DPT		:= 76, 
            typDPT			  := PersistentVars.typDPT[2][76], 
        );

        
                                    
        C_5640_501_06_KAB6020_A1_R0543.xIn := M2_076_543_KAB6020_POS_ACT.xTimeOut;
                                    
        M2_077_543_KAB6021_CV(
            bPortKNX		  := 2, 
            dwIndex_DPT		:= 77, 
            typDPT			  := PersistentVars.typDPT[2][77],
            xUpdate_KNX		:= PRG_KnxMaster.updateHeat, 
        );

        M2_077_543_KAB6021_CV.rValue_IN := GVL_ClimateControl.typClimateControllerInterfaceRoom543.actuators.heating.controlledVariable;        
         
        M2_078_543_KAB6021_POS_ACT(
            bPortKNX		   := 2, 
            dwIndex_DPT		:= 78, 
            typDPT			  := PersistentVars.typDPT[2][78], 
        );

        
                                    
        C_5640_501_06_KAB6021_A1_R0543.xIn := M2_078_543_KAB6021_POS_ACT.xTimeOut;
                                    
        M2_079_547_1_KAB6022_CV(
            bPortKNX		  := 2, 
            dwIndex_DPT		:= 79, 
            typDPT			  := PersistentVars.typDPT[2][79],
            xUpdate_KNX		:= PRG_KnxMaster.updateHeat, 
        );

        M2_079_547_1_KAB6022_CV.rValue_IN := GVL_ClimateControl.typClimateControllerInterfaceRoom547_1.actuators.heating.controlledVariable;        
         
        M2_080_547_1_KAB6022_POS_ACT(
            bPortKNX		   := 2, 
            dwIndex_DPT		:= 80, 
            typDPT			  := PersistentVars.typDPT[2][80], 
        );

        
                                    
        C_5640_501_06_KAB6022_A1_R0547_1.xIn := M2_080_547_1_KAB6022_POS_ACT.xTimeOut;
                                    
        M2_081_547_1_KAB6023_CV(
            bPortKNX		  := 2, 
            dwIndex_DPT		:= 81, 
            typDPT			  := PersistentVars.typDPT[2][81],
            xUpdate_KNX		:= PRG_KnxMaster.updateHeat, 
        );

        M2_081_547_1_KAB6023_CV.rValue_IN := GVL_ClimateControl.typClimateControllerInterfaceRoom547_1.actuators.heating.controlledVariable;        
         
        M2_082_547_1_KAB6023_POS_ACT(
            bPortKNX		   := 2, 
            dwIndex_DPT		:= 82, 
            typDPT			  := PersistentVars.typDPT[2][82], 
        );

        
                                    
        C_5640_501_06_KAB6023_A1_R0547_1.xIn := M2_082_547_1_KAB6023_POS_ACT.xTimeOut;
                                    
        M2_083_547_1_KAB6024_CV(
            bPortKNX		  := 2, 
            dwIndex_DPT		:= 83, 
            typDPT			  := PersistentVars.typDPT[2][83],
            xUpdate_KNX		:= PRG_KnxMaster.updateHeat, 
        );

        M2_083_547_1_KAB6024_CV.rValue_IN := GVL_ClimateControl.typClimateControllerInterfaceRoom547_1.actuators.heating.controlledVariable;        
         
        M2_084_547_1_KAB6024_POS_ACT(
            bPortKNX		   := 2, 
            dwIndex_DPT		:= 84, 
            typDPT			  := PersistentVars.typDPT[2][84], 
        );

        
                                    
        C_5640_501_06_KAB6024_A1_R0547_1.xIn := M2_084_547_1_KAB6024_POS_ACT.xTimeOut;
                                    
        M2_085_547_2_KAB6025_CV(
            bPortKNX		  := 2, 
            dwIndex_DPT		:= 85, 
            typDPT			  := PersistentVars.typDPT[2][85],
            xUpdate_KNX		:= PRG_KnxMaster.updateHeat, 
        );

        M2_085_547_2_KAB6025_CV.rValue_IN := GVL_ClimateControl.typClimateControllerInterfaceRoom547_2.actuators.heating.controlledVariable;        
         
        M2_086_547_2_KAB6025_POS_ACT(
            bPortKNX		   := 2, 
            dwIndex_DPT		:= 86, 
            typDPT			  := PersistentVars.typDPT[2][86], 
        );

        
                                    
        C_5640_501_06_KAB6025_A1_R0547_2.xIn := M2_086_547_2_KAB6025_POS_ACT.xTimeOut;
                                    
        M2_087_547_2_KAB6026_CV(
            bPortKNX		  := 2, 
            dwIndex_DPT		:= 87, 
            typDPT			  := PersistentVars.typDPT[2][87],
            xUpdate_KNX		:= PRG_KnxMaster.updateHeat, 
        );

        M2_087_547_2_KAB6026_CV.rValue_IN := GVL_ClimateControl.typClimateControllerInterfaceRoom547_2.actuators.heating.controlledVariable;        
         
        M2_088_547_2_KAB6026_POS_ACT(
            bPortKNX		   := 2, 
            dwIndex_DPT		:= 88, 
            typDPT			  := PersistentVars.typDPT[2][88], 
        );

        
                                    
        C_5640_501_06_KAB6026_A1_R0547_2.xIn := M2_088_547_2_KAB6026_POS_ACT.xTimeOut;
                                    
        M2_089_547_2_KAB6027_CV(
            bPortKNX		  := 2, 
            dwIndex_DPT		:= 89, 
            typDPT			  := PersistentVars.typDPT[2][89],
            xUpdate_KNX		:= PRG_KnxMaster.updateHeat, 
        );

        M2_089_547_2_KAB6027_CV.rValue_IN := GVL_ClimateControl.typClimateControllerInterfaceRoom547_2.actuators.heating.controlledVariable;        
         
        M2_090_547_2_KAB6027_POS_ACT(
            bPortKNX		   := 2, 
            dwIndex_DPT		:= 90, 
            typDPT			  := PersistentVars.typDPT[2][90], 
        );

        
                                    
        C_5640_501_06_KAB6027_A1_R0547_2.xIn := M2_090_547_2_KAB6027_POS_ACT.xTimeOut;
                                    
        M2_091_544_KAB6028_CV(
            bPortKNX		  := 2, 
            dwIndex_DPT		:= 91, 
            typDPT			  := PersistentVars.typDPT[2][91],
            xUpdate_KNX		:= PRG_KnxMaster.updateHeat, 
        );

        M2_091_544_KAB6028_CV.rValue_IN := GVL_ClimateControl.typClimateControllerInterfaceRoom544.actuators.heating.controlledVariable;        
         
        M2_092_544_KAB6028_POS_ACT(
            bPortKNX		   := 2, 
            dwIndex_DPT		:= 92, 
            typDPT			  := PersistentVars.typDPT[2][92], 
        );

        
                                    
        C_5640_501_06_KAB6028_A1_R0544.xIn := M2_092_544_KAB6028_POS_ACT.xTimeOut;
                                    
                
              
END_PROGRAM

PROGRAM PRG_DamperLine_1

                
    
	if (firstScan) then
	    initialSettings();
	end_if
	
	GVL_Modbus.modbusDamperInterface[1][1].tag     := 'A=360.01-SQ4A407';
	GVL_Modbus.modbusDamperInterface[1][2].tag     := 'A=360.01-SQ44AH2';
	GVL_Modbus.modbusDamperInterface[1][3].tag     := 'A=360.01-SQ44AH1';
	GVL_Modbus.modbusDamperInterface[1][4].tag     := 'A=360.01-SQ54AH1';
	GVL_Modbus.modbusDamperInterface[1][5].tag     := 'A=360.01-SQ5A405';
	GVL_Modbus.modbusDamperInterface[1][6].tag     := 'A=360.01-SQ4A401_2';
	GVL_Modbus.modbusDamperInterface[1][7].tag     := 'A=360.01-SQ4A401_1';
	GVL_Modbus.modbusDamperInterface[1][8].tag     := 'A=360.01-SQ4A401';
	GVL_Modbus.modbusDamperInterface[1][9].tag     := 'A=360.01-SQ4A406';
	GVL_Modbus.modbusDamperInterface[1][10].tag     := 'A=360.01-SQ4A408';
	GVL_Modbus.modbusDamperInterface[1][11].tag     := 'A=360.01-SQ4A410_1';
	GVL_Modbus.modbusDamperInterface[1][12].tag     := 'A=360.01-SQ4A410_2';
	GVL_Modbus.modbusDamperInterface[1][13].tag     := 'A=360.01-SQ4A410_3';
	GVL_Modbus.modbusDamperInterface[1][14].tag     := 'A=360.01-SQ4A410_4';
	GVL_Modbus.modbusDamperInterface[1][15].tag     := 'A=360.01-SQ4A410_5';
	GVL_Modbus.modbusDamperInterface[1][16].tag     := 'A=360.01-SQ4A412';
	GVL_Modbus.modbusDamperInterface[1][17].tag     := 'A=360.01-SQ4A413';
	GVL_Modbus.modbusDamperInterface[1][18].tag     := 'A=360.01-SK4A415';
	GVL_Modbus.modbusDamperInterface[1][19].tag     := 'A=360.01-SK5A415';
	GVL_Modbus.modbusDamperInterface[1][20].tag     := 'A=360.01-SK5A418';
	GVL_Modbus.modbusDamperInterface[1][21].tag     := 'A=360.01-SK4A417';
	GVL_Modbus.modbusDamperInterface[1][22].tag     := 'A=360.01-SQ5C411';
	GVL_Modbus.modbusDamperInterface[1][1].damperClimateInterface     := GVL_ClimateControl.typClimateControllerInterfaceRoomA407.actuators.damper;
	GVL_Modbus.modbusDamperInterface[1][2].damperClimateInterface     := GVL_ClimateControl.typClimateControllerInterfaceRoomSONE.actuators.damper;
	GVL_Modbus.modbusDamperInterface[1][3].damperClimateInterface     := GVL_ClimateControl.typClimateControllerInterfaceRoomSONE.actuators.damper;
	GVL_Modbus.modbusDamperInterface[1][4].damperClimateInterface     := GVL_ClimateControl.typClimateControllerInterfaceRoomSONE.actuators.damper;
	GVL_Modbus.modbusDamperInterface[1][5].damperClimateInterface     := GVL_ClimateControl.typClimateControllerInterfaceRoomA405.actuators.damper;
	GVL_Modbus.modbusDamperInterface[1][6].damperClimateInterface     := GVL_ClimateControl.typClimateControllerInterfaceRoomA401_4.actuators.damper;
	GVL_Modbus.modbusDamperInterface[1][7].damperClimateInterface     := GVL_ClimateControl.typClimateControllerInterfaceRoomA401_4.actuators.damper;
	GVL_Modbus.modbusDamperInterface[1][8].damperClimateInterface     := GVL_ClimateControl.typClimateControllerInterfaceRoomA401_4.actuators.damper;
	GVL_Modbus.modbusDamperInterface[1][9].damperClimateInterface     := GVL_ClimateControl.typClimateControllerInterfaceRoomA406.actuators.damper;
	GVL_Modbus.modbusDamperInterface[1][10].damperClimateInterface     := GVL_ClimateControl.typClimateControllerInterfaceRoomA408.actuators.damper;
	GVL_Modbus.modbusDamperInterface[1][11].damperClimateInterface     := GVL_ClimateControl.typClimateControllerInterfaceRoomA410_1.actuators.damper;
	GVL_Modbus.modbusDamperInterface[1][12].damperClimateInterface     := GVL_ClimateControl.typClimateControllerInterfaceRoomA410_1.actuators.damper;
	GVL_Modbus.modbusDamperInterface[1][13].damperClimateInterface     := GVL_ClimateControl.typClimateControllerInterfaceRoomA410_1.actuators.damper;
	GVL_Modbus.modbusDamperInterface[1][14].damperClimateInterface     := GVL_ClimateControl.typClimateControllerInterfaceRoomA410_2.actuators.damper;
	GVL_Modbus.modbusDamperInterface[1][15].damperClimateInterface     := GVL_ClimateControl.typClimateControllerInterfaceRoomA410_2.actuators.damper;
	GVL_Modbus.modbusDamperInterface[1][16].damperClimateInterface     := GVL_ClimateControl.typClimateControllerInterfaceRoomA412.actuators.damper;
	GVL_Modbus.modbusDamperInterface[1][17].damperClimateInterface     := GVL_ClimateControl.typClimateControllerInterfaceRoomA413.actuators.damper;
	GVL_Modbus.modbusDamperInterface[1][18].damperClimateInterface.setpoint     := 100;
	GVL_Modbus.modbusDamperInterface[1][19].damperClimateInterface.setpoint     := 100;
	GVL_Modbus.modbusDamperInterface[1][20].damperClimateInterface.setpoint     := 100;
	GVL_Modbus.modbusDamperInterface[1][21].damperClimateInterface.setpoint     := 100;
	GVL_Modbus.modbusDamperInterface[1][22].damperClimateInterface     := GVL_ClimateControl.typClimateControllerInterfaceRoomC411.actuators.damper;
                
              

ACTION initialSettings:
                            
                                
	GVL_Modbus.modbusDamperInterface[1][1].enable     := TRUE;
	GVL_Modbus.modbusDamperInterface[1][2].enable     := TRUE;
	GVL_Modbus.modbusDamperInterface[1][3].enable     := TRUE;
	GVL_Modbus.modbusDamperInterface[1][4].enable     := TRUE;
	GVL_Modbus.modbusDamperInterface[1][5].enable     := TRUE;
	GVL_Modbus.modbusDamperInterface[1][6].enable     := TRUE;
	GVL_Modbus.modbusDamperInterface[1][7].enable     := TRUE;
	GVL_Modbus.modbusDamperInterface[1][8].enable     := TRUE;
	GVL_Modbus.modbusDamperInterface[1][9].enable     := TRUE;
	GVL_Modbus.modbusDamperInterface[1][10].enable     := TRUE;
	GVL_Modbus.modbusDamperInterface[1][11].enable     := TRUE;
	GVL_Modbus.modbusDamperInterface[1][12].enable     := TRUE;
	GVL_Modbus.modbusDamperInterface[1][13].enable     := TRUE;
	GVL_Modbus.modbusDamperInterface[1][14].enable     := TRUE;
	GVL_Modbus.modbusDamperInterface[1][15].enable     := TRUE;
	GVL_Modbus.modbusDamperInterface[1][16].enable     := TRUE;
	GVL_Modbus.modbusDamperInterface[1][17].enable     := TRUE;
	GVL_Modbus.modbusDamperInterface[1][18].enable     := TRUE;
	GVL_Modbus.modbusDamperInterface[1][19].enable     := TRUE;
	GVL_Modbus.modbusDamperInterface[1][20].enable     := TRUE;
	GVL_Modbus.modbusDamperInterface[1][21].enable     := TRUE;
	GVL_Modbus.modbusDamperInterface[1][22].enable     := TRUE;
	GVL_Modbus.modbusDamperInterface[1][1].systemNumber     := 01;
	GVL_Modbus.modbusDamperInterface[1][2].systemNumber     := 01;
	GVL_Modbus.modbusDamperInterface[1][3].systemNumber     := 01;
	GVL_Modbus.modbusDamperInterface[1][4].systemNumber     := 01;
	GVL_Modbus.modbusDamperInterface[1][5].systemNumber     := 01;
	GVL_Modbus.modbusDamperInterface[1][6].systemNumber     := 01;
	GVL_Modbus.modbusDamperInterface[1][7].systemNumber     := 01;
	GVL_Modbus.modbusDamperInterface[1][8].systemNumber     := 01;
	GVL_Modbus.modbusDamperInterface[1][9].systemNumber     := 01;
	GVL_Modbus.modbusDamperInterface[1][10].systemNumber     := 01;
	GVL_Modbus.modbusDamperInterface[1][11].systemNumber     := 01;
	GVL_Modbus.modbusDamperInterface[1][12].systemNumber     := 01;
	GVL_Modbus.modbusDamperInterface[1][13].systemNumber     := 01;
	GVL_Modbus.modbusDamperInterface[1][14].systemNumber     := 01;
	GVL_Modbus.modbusDamperInterface[1][15].systemNumber     := 01;
	GVL_Modbus.modbusDamperInterface[1][16].systemNumber     := 01;
	GVL_Modbus.modbusDamperInterface[1][17].systemNumber     := 01;
	GVL_Modbus.modbusDamperInterface[1][18].systemNumber     := 01;
	GVL_Modbus.modbusDamperInterface[1][19].systemNumber     := 01;
	GVL_Modbus.modbusDamperInterface[1][20].systemNumber     := 01;
	GVL_Modbus.modbusDamperInterface[1][21].systemNumber     := 01;
	GVL_Modbus.modbusDamperInterface[1][22].systemNumber     := 01;
	GVL_Modbus.modbusDamperInterface[1][1].systemPrefix     := 'A';
	GVL_Modbus.modbusDamperInterface[1][2].systemPrefix     := 'A';
	GVL_Modbus.modbusDamperInterface[1][3].systemPrefix     := 'A';
	GVL_Modbus.modbusDamperInterface[1][4].systemPrefix     := 'A';
	GVL_Modbus.modbusDamperInterface[1][5].systemPrefix     := 'A';
	GVL_Modbus.modbusDamperInterface[1][6].systemPrefix     := 'A';
	GVL_Modbus.modbusDamperInterface[1][7].systemPrefix     := 'A';
	GVL_Modbus.modbusDamperInterface[1][8].systemPrefix     := 'A';
	GVL_Modbus.modbusDamperInterface[1][9].systemPrefix     := 'A';
	GVL_Modbus.modbusDamperInterface[1][10].systemPrefix     := 'A';
	GVL_Modbus.modbusDamperInterface[1][11].systemPrefix     := 'A';
	GVL_Modbus.modbusDamperInterface[1][12].systemPrefix     := 'A';
	GVL_Modbus.modbusDamperInterface[1][13].systemPrefix     := 'A';
	GVL_Modbus.modbusDamperInterface[1][14].systemPrefix     := 'A';
	GVL_Modbus.modbusDamperInterface[1][15].systemPrefix     := 'A';
	GVL_Modbus.modbusDamperInterface[1][16].systemPrefix     := 'A';
	GVL_Modbus.modbusDamperInterface[1][17].systemPrefix     := 'A';
	GVL_Modbus.modbusDamperInterface[1][18].systemPrefix     := 'A';
	GVL_Modbus.modbusDamperInterface[1][19].systemPrefix     := 'A';
	GVL_Modbus.modbusDamperInterface[1][20].systemPrefix     := 'A';
	GVL_Modbus.modbusDamperInterface[1][21].systemPrefix     := 'A';
	GVL_Modbus.modbusDamperInterface[1][22].systemPrefix     := 'A';
	GVL_Modbus.modbusDamperInterface[1][1].airDirection     := 0;
	GVL_Modbus.modbusDamperInterface[1][2].airDirection     := 0;
	GVL_Modbus.modbusDamperInterface[1][3].airDirection     := 0;
	GVL_Modbus.modbusDamperInterface[1][4].airDirection     := 1;
	GVL_Modbus.modbusDamperInterface[1][5].airDirection     := 1;
	GVL_Modbus.modbusDamperInterface[1][6].airDirection     := 0;
	GVL_Modbus.modbusDamperInterface[1][7].airDirection     := 0;
	GVL_Modbus.modbusDamperInterface[1][8].airDirection     := 0;
	GVL_Modbus.modbusDamperInterface[1][9].airDirection     := 0;
	GVL_Modbus.modbusDamperInterface[1][10].airDirection     := 0;
	GVL_Modbus.modbusDamperInterface[1][11].airDirection     := 0;
	GVL_Modbus.modbusDamperInterface[1][12].airDirection     := 0;
	GVL_Modbus.modbusDamperInterface[1][13].airDirection     := 0;
	GVL_Modbus.modbusDamperInterface[1][14].airDirection     := 0;
	GVL_Modbus.modbusDamperInterface[1][15].airDirection     := 0;
	GVL_Modbus.modbusDamperInterface[1][16].airDirection     := 0;
	GVL_Modbus.modbusDamperInterface[1][17].airDirection     := 0;
	GVL_Modbus.modbusDamperInterface[1][18].airDirection     := 1;
	GVL_Modbus.modbusDamperInterface[1][19].airDirection     := 1;
	GVL_Modbus.modbusDamperInterface[1][20].airDirection     := 1;
	GVL_Modbus.modbusDamperInterface[1][21].airDirection     := 1;
	GVL_Modbus.modbusDamperInterface[1][22].airDirection     := 1;
	PersistentVars.ModbusDamperSetpoints[1][1].vMidM3h     := 490;
	PersistentVars.ModbusDamperSetpoints[1][6].vMidM3h     := 100;
	PersistentVars.ModbusDamperSetpoints[1][7].vMidM3h     := 100;
	PersistentVars.ModbusDamperSetpoints[1][8].vMidM3h     := 100;
	PersistentVars.ModbusDamperSetpoints[1][9].vMidM3h     := 100;
	PersistentVars.ModbusDamperSetpoints[1][10].vMidM3h     := 160;
	PersistentVars.ModbusDamperSetpoints[1][11].vMidM3h     := 100;
	PersistentVars.ModbusDamperSetpoints[1][12].vMidM3h     := 100;
	PersistentVars.ModbusDamperSetpoints[1][13].vMidM3h     := 100;
	PersistentVars.ModbusDamperSetpoints[1][14].vMidM3h     := 100;
	PersistentVars.ModbusDamperSetpoints[1][15].vMidM3h     := 100;
	PersistentVars.ModbusDamperSetpoints[1][16].vMidM3h     := 100;
	PersistentVars.ModbusDamperSetpoints[1][17].vMidM3h     := 340;
                            
                        
END_ACTION
END_PROGRAM

PROGRAM PRG_DamperLine_2

                
    
	if (firstScan) then
	    initialSettings();
	end_if
	
	GVL_Modbus.modbusDamperInterface[2][1].tag     := 'A=360.01-SK5A421';
	GVL_Modbus.modbusDamperInterface[2][2].tag     := 'A=360.01-SQ54AH2';
	GVL_Modbus.modbusDamperInterface[2][3].tag     := 'A=360.01-SK5A424';
	GVL_Modbus.modbusDamperInterface[2][4].tag     := 'A=360.01-SQ44AH3';
	GVL_Modbus.modbusDamperInterface[2][5].tag     := 'A=360.01-SQ44AH4';
	GVL_Modbus.modbusDamperInterface[2][6].tag     := 'A=360.01-SQ44AH5';
	GVL_Modbus.modbusDamperInterface[2][7].tag     := 'A=360.01-SQ54AH3';
	GVL_Modbus.modbusDamperInterface[2][8].tag     := 'A=360.01-SQ5A401';
	GVL_Modbus.modbusDamperInterface[2][9].tag     := 'A=360.01-SQ4A403';
	GVL_Modbus.modbusDamperInterface[2][10].tag     := 'A=360.01-SQ4A401_3';
	GVL_Modbus.modbusDamperInterface[2][11].tag     := 'A=360.01-SQ4A401_4';
	GVL_Modbus.modbusDamperInterface[2][12].tag     := 'A=360.01-SQ4A401_5';
	GVL_Modbus.modbusDamperInterface[2][13].tag     := 'A=360.01-SQ4A401_6';
	GVL_Modbus.modbusDamperInterface[2][14].tag     := 'A=360.01-SQ4A401_7';
	GVL_Modbus.modbusDamperInterface[2][15].tag     := 'A=360.01-SQ4A401_8';
	GVL_Modbus.modbusDamperInterface[2][16].tag     := 'A=360.01-SQ4A401_9';
	GVL_Modbus.modbusDamperInterface[2][17].tag     := 'A=360.01-SQ4A401_0';
	GVL_Modbus.modbusDamperInterface[2][18].tag     := 'A=360.01-SQ4A426';
	GVL_Modbus.modbusDamperInterface[2][19].tag     := 'A=360.01-SQ4A428_1';
	GVL_Modbus.modbusDamperInterface[2][20].tag     := 'A=360.01-SQ4A428_2';
	GVL_Modbus.modbusDamperInterface[2][21].tag     := 'A=360.01-SQ4A428_3';
	GVL_Modbus.modbusDamperInterface[2][22].tag     := 'A=360.01-SQ4A428_4';
	GVL_Modbus.modbusDamperInterface[2][23].tag     := 'A=360.01-SQ5A425';
	GVL_Modbus.modbusDamperInterface[2][24].tag     := 'A=360.01-SQ4A428_5';
	GVL_Modbus.modbusDamperInterface[2][25].tag     := 'A=360.01-SQ4A428_6';
	GVL_Modbus.modbusDamperInterface[2][26].tag     := 'A=360.01-SQ4A428_7';
	GVL_Modbus.modbusDamperInterface[2][1].damperClimateInterface.setpoint     := 100;
	GVL_Modbus.modbusDamperInterface[2][2].damperClimateInterface     := GVL_ClimateControl.typClimateControllerInterfaceRoomSONE.actuators.damper;
	GVL_Modbus.modbusDamperInterface[2][3].damperClimateInterface     := GVL_ClimateControl.typClimateControllerInterfaceRoomA424.actuators.damper;
	GVL_Modbus.modbusDamperInterface[2][4].damperClimateInterface     := GVL_ClimateControl.typClimateControllerInterfaceRoomSONE.actuators.damper;
	GVL_Modbus.modbusDamperInterface[2][5].damperClimateInterface     := GVL_ClimateControl.typClimateControllerInterfaceRoomSONE.actuators.damper;
	GVL_Modbus.modbusDamperInterface[2][6].damperClimateInterface     := GVL_ClimateControl.typClimateControllerInterfaceRoomSONE.actuators.damper;
	GVL_Modbus.modbusDamperInterface[2][7].damperClimateInterface     := GVL_ClimateControl.typClimateControllerInterfaceRoomSONE.actuators.damper;
	GVL_Modbus.modbusDamperInterface[2][8].damperClimateInterface     := GVL_ClimateControl.typClimateControllerInterfaceRoomA401.actuators.damper;
	GVL_Modbus.modbusDamperInterface[2][9].damperClimateInterface     := GVL_ClimateControl.typClimateControllerInterfaceRoomA403.actuators.damper;
	GVL_Modbus.modbusDamperInterface[2][10].damperClimateInterface     := GVL_ClimateControl.typClimateControllerInterfaceRoomA401_3.actuators.damper;
	GVL_Modbus.modbusDamperInterface[2][11].damperClimateInterface     := GVL_ClimateControl.typClimateControllerInterfaceRoomA401_3.actuators.damper;
	GVL_Modbus.modbusDamperInterface[2][12].damperClimateInterface     := GVL_ClimateControl.typClimateControllerInterfaceRoomA401_2.actuators.damper;
	GVL_Modbus.modbusDamperInterface[2][13].damperClimateInterface     := GVL_ClimateControl.typClimateControllerInterfaceRoomA401_2.actuators.damper;
	GVL_Modbus.modbusDamperInterface[2][14].damperClimateInterface     := GVL_ClimateControl.typClimateControllerInterfaceRoomA401_2.actuators.damper;
	GVL_Modbus.modbusDamperInterface[2][15].damperClimateInterface     := GVL_ClimateControl.typClimateControllerInterfaceRoomA401_1.actuators.damper;
	GVL_Modbus.modbusDamperInterface[2][16].damperClimateInterface     := GVL_ClimateControl.typClimateControllerInterfaceRoomA401_1.actuators.damper;
	GVL_Modbus.modbusDamperInterface[2][17].damperClimateInterface     := GVL_ClimateControl.typClimateControllerInterfaceRoomA401_1.actuators.damper;
	GVL_Modbus.modbusDamperInterface[2][18].damperClimateInterface     := GVL_ClimateControl.typClimateControllerInterfaceRoomA426.actuators.damper;
	GVL_Modbus.modbusDamperInterface[2][19].damperClimateInterface     := GVL_ClimateControl.typClimateControllerInterfaceRoomA428_3.actuators.damper;
	GVL_Modbus.modbusDamperInterface[2][20].damperClimateInterface     := GVL_ClimateControl.typClimateControllerInterfaceRoomA428_3.actuators.damper;
	GVL_Modbus.modbusDamperInterface[2][21].damperClimateInterface     := GVL_ClimateControl.typClimateControllerInterfaceRoomA428_3.actuators.damper;
	GVL_Modbus.modbusDamperInterface[2][22].damperClimateInterface     := GVL_ClimateControl.typClimateControllerInterfaceRoomA428_2.actuators.damper;
	GVL_Modbus.modbusDamperInterface[2][23].damperClimateInterface     := GVL_ClimateControl.typClimateControllerInterfaceRoomA425.actuators.damper;
	GVL_Modbus.modbusDamperInterface[2][24].damperClimateInterface     := GVL_ClimateControl.typClimateControllerInterfaceRoomA428_2.actuators.damper;
	GVL_Modbus.modbusDamperInterface[2][25].damperClimateInterface     := GVL_ClimateControl.typClimateControllerInterfaceRoomA428_1.actuators.damper;
	GVL_Modbus.modbusDamperInterface[2][26].damperClimateInterface     := GVL_ClimateControl.typClimateControllerInterfaceRoomA428_1.actuators.damper;
                
              

ACTION initialSettings:
                            
                                
